(* IEC 61131-3 sources: sistemas-de-automacao/, 39 files *)

(* ---- E_PRODUCT_TYPE (DUT).st ---- *)
{attribute 'qualified_only'}
{attribute 'strict'}

// Enum para os tipos de itens que podem ser gerados e identificados no início da operação

TYPE E_PRODUCT_TYPE :
(
	e_productType_unknown := 0, // Caso o item ainda não tenha sido identificado ou tenha ocorrido algum erro
								// durante a identificação
	e_productType_plastic := 1, // Caso o item seja um bloco de plástico
	e_productType_metal := 2, // Caso o item seja um bloco de metal
	e_productType_box := 3 // Caso o item seja uma caixa
);
END_TYPE

(* ---- ST_PRODUCT (DUT).st ---- *)
TYPE ST_PRODUCT :

// Struct que guarda as informações sobre um produto, como o tipo dele, se ele já foi processado ou se ele é metálico
// Na prática só foi usada a informação de se o produto é metálico ou não, mas caso o projeto necessitasse de mais
// features ou fosse expandido de alguma forma, a struct permitiria essas expansão sem muito retrabalho

STRUCT
	productType : E_PRODUCT_TYPE;
	processed : BOOL;
	metal : BOOL;
END_STRUCT
END_TYPE

(* ---- ST_PRODUCT.DUT ---- *)
TYPE ST_PRODUCT :
STRUCT
	productType : E_PRODUCT_TYPE;
	metal       :           BOOL;
	processed   :           BOOL;

END_STRUCT
END_TYPE

(* ---- ST_PRODUCT.st ---- *)
TYPE ST_PRODUCT :
STRUCT
	productType : E_PRODUCT_TYPE;
	processed : BOOL;

END_STRUCT
END_TYPE

(* ---- ST_QUEUE.st ---- *)
TYPE ST_QUEUE :
STRUCT
 head : POINTER OF ST_QUEUE_ITEM;
 tail : POINTER OF ST_QUEUE_ITEM;
END_STRUCT
END_TYPE

(* ---- constante (GVL).st ---- *)
VAR_GLOBAL CONSTANT
    Xidle : INT := 500; // As coordenadas do Gantry CNC quando ele estiver ocioso
    Yidle : INT := 500;
    Zidle : INT := 200;

    XconveyorPlas : INT := 470; // As coordenadas do Gantry CNC para detectar uma caixa passando
    YconveyorPlas : INT := 600; // pela esteira de plástico usando o sensor SPP
    ZconveyorPlas : INT := 1000;

    XconveyorMetal : INT := 1000; // As coordenadas do Gantry CNC para detectar uma caixa passando
    YconveyorMetal : INT := 600;  // pela esteira de plástico usando o sensor SPP
    ZconveyorMetal : INT := 1000;

    Xpart : INT := 110; // As coordenadas do Gantry CNC para pegar uma peça na esteira da usinagem
    Ypart : INT := 500;
    Zpart : INT := 830;

    XboxMetal : INT := 850; // As coordenadas do Gantry CNC para pôr uma peça numa caixa da esteira
    YboxMetal : INT := 500; // de metal
    ZboxMetal : INT := 800;

    XboxPlas : INT := 330; // As coordenadas do Gantry CNC para pôr uma peça numa caixa da esteira
    YboxPlas : INT := 500; // de plástico
    ZboxPlas : INT := 800;

END_VAR

(* ---- constante.VAR ---- *)
{attribute 'qualified_only'}
VAR_GLOBAL CONSTANT
    Xidle : INT := 500;
    Yidle : INT := 500;
    Zidle : INT := 200;

    XconveyorPlas : INT := 470;
    YconveyorPlas : INT := 600;
    ZconveyorPlas : INT := 1000;

    XconveyorMetal : INT := 1000;
    YconveyorMetal : INT := 600;
    ZconveyorMetal : INT := 1000;

    Xpart : INT := 110;
    Ypart : INT := 500;
    Zpart : INT := 830;

    XboxMetal : INT := 850;
    YboxMetal : INT := 500;
    ZboxMetal : INT := 800;

    XboxPlas : INT := 330;
    YboxPlas : INT := 500;
    ZboxPlas : INT := 800;

END_VAR

(* ---- FIO (GVL).st ---- *)
{attribute 'qualified_only'}
VAR_GLOBAL
    i_DS2        			  		: BOOL; // Sensor óptico da balança
    i_Emergencia              		: BOOL; // Botão de emergência
	i_MachiningCenterOpened   		: BOOL; // Centro de usinagem livre
	i_MachiningCenterIsBusy   		: BOOL; // Centro de usinagem trabalhando
	i_MachiningCenterHasError 		: BOOL; // Erro no processo de usinagem
	i_RS1 					  		: BOOL; // Sensor óptico da usinagem
	i_RS2 					  		: BOOL; // Sensor óptico do empacotamento
	i_SC    				  		: BOOL; // Sensor capacitivo
	i_SC1Mais 				  		: BOOL; // Fim de curso do pistão - estendido
	i_SC1Menos 	 			  		: BOOL; // Fim de curso do pistão - retraido
    i_SI        			  		: BOOL; // Sensor indutivo
	i_SP 					  		:  INT; // Sensor da balança (4.0 plástico; 5.0 metal; 1.5 caixa)
	i_SPMais 				  		: BOOL; // Botão de aumentar quantidade de itens por caixa
	i_SPMenos 				  		: BOOL; // Botão de diminuir quantidade de itens por caixa
	i_SPP 					  		: BOOL; // Sensor de item pego pela ponte CNC
	i_Start 				  		: BOOL; // Botão START
	i_Stop 					  		: BOOL; // Botão STOP
    i_XPOS        			  		:  INT; // Dado da posição X atual da ponte CNC
    i_YPOS    				  		:  INT; // Dado da posição Y atual da ponte CNC
    i_ZPOS      			  		:  INT; // Dado da posição Z atual da ponte CNC
	i_DS3        			  		: BOOL; // Sensor óptico da esteira de plástico
	i_DS4        			  		: BOOL; // Sensor óptico da esteira de metal

	o_C1 					  		: BOOL; // Pistão
	o_Caixas_Emissor_1 		  		: BOOL; // Emissor de caixas (metal)
	o_E1 					  		: BOOL; // Primeira Esteira do classificador
	o_E2 					  		: BOOL; // Esteira final do classificador e inicial da usinagem
	o_E3 					  		: BOOL; // Esteira inicial do empacotamento
	o_EMETAL1 				  		: BOOL; // Primeira esteira de rolo do empacotamento de metal
	o_EMETAL2 				  		: BOOL; // Segunda esteira de rolo do empacotamento de metal
	o_EMETAL3 				  		: BOOL; // Terceira esteira de rolo do empacotamento de metal
	o_Emissor_Partes 		  		: BOOL; // Emissor dos itens (Deixar ligado)
	o_Emitter_4 			  		: BOOL; // Emissor de caixas (plástico)
	o_EPLASTIC1 			  		: BOOL; // Primeira esteira de rolo do empacotamento de plástico
	o_EPLASTIC2 			  		: BOOL; // Segunda esteira de rolo do empacotamento de plástico
	o_EPLASTIC3 			  	   	: BOOL; // Terceira esteira de rolo do empacotamento de plástico
	o_E_SP 					  	   	: BOOL; // Esteira da balança
	o_LedG 					  	   	: BOOL; // Led verde no canto da usinagem
	o_LedR 					  	   	: BOOL; // Led vermelho no canto da usinagem
	o_LedSPMais 			  	   	: BOOL; // Led do botão SP+
	o_LedSPMenos 			  	   	: BOOL; // Led do botão SP-
	o_LedStart 				  	   	: BOOL; // Led do botão START
	o_LedStop 				  	   	: BOOL; // Led do botão STOP
	o_LedY 					  	   	: BOOL; // Led amarelo no canto da usinagem
    o_RB1_Stop 				  	   	: BOOL; // Botão de interrupção do processo do braço robótico + usinagem
	o_RB1_Reset 			  	   	: BOOL; // Botão de reset do processo do braço robótico + usinagem
	o_RB1_Start 			  	  	: BOOL; // Botão de iniciar o processo do braço robótico + usinagem
	o_Succao 				  	  	: BOOL; // Acionamento da sucção da ponte CNC
    o_X           			  		:  INT; // Posição X da ponte CNC
    o_Y   					  		:  INT; // Posição Y da ponte CNC
    o_Z  					  		:  INT; // Posição Z da ponte CNC
	o_MachiningCenterProduceLids    : BOOL; // Modo de usinagem do plástico
	o_NumCaixas               		:  INT;  // Número de caixas
	o_NumMetal                		:  INT;  // Número de itens de metal
	o_NumPlastico             		:  INT;  // Número de itens de plástico
END_VAR

(* ---- FIO.VAR ---- *)
{attribute 'qualified_only'}
VAR_GLOBAL
    i_DS2        			  : BOOL; // Sensor óptico da balança
    i_Emergencia              : BOOL; // Botão de emergência
	i_MachiningCenterOpened   : BOOL; // Centro de usinagem livre
	i_MachiningCenterIsBusy   : BOOL; // Centro de usinagem trabalhando
	i_MachiningCenterHasError : BOOL; // Erro no processo de usinagem
	i_RS1 					  : BOOL; // Sensor óptico da usinagem
	i_RS2 					  : BOOL; // Sensor óptico do empacotamento
	i_SC    				  : BOOL; // Sensor capacitivo
	i_SC1Mais 				  : BOOL; // Fim de curso do pistão - estendido
	i_SC1Menos 	 			  : BOOL; // Fim de curso do pistão - retraido
    i_SI        			  : BOOL; // Sensor indutivo
	i_SP 					  : REAL; // Sensor da balança (4.0 plástico; 5.0 metal; 1.5 caixa)
	i_SPMais 				  : BOOL; // Botão de aumentar quantidade de itens por caixa
	i_SPMenos 				  : BOOL; // Botão de diminuir quantidade de itens por caixa
	i_SPP 					  : BOOL; // Sensor de item pego pela ponte CNC
	i_Start 				  : BOOL; // Botão START
	i_Stop 					  : BOOL; // Botão STOP
    i_XPOS        			  : REAL; // Dado da posição X atual da ponte CNC
    i_YPOS    				  : REAL; // Dado da posição Y atual da ponte CNC
    i_ZPOS      			  : REAL; // Dado da posição Z atual da ponte CNC

	o_C1 					  : BOOL; // Pistão
	o_Caixas_Emissor_1 		  : BOOL; // Emissor de caixas (metal)
	o_E1 					  : BOOL; // Primeira Esteira do classificador
	o_E2 					  : BOOL; // Esteira final do classificador e inicial da usinagem
	o_E3 					  : BOOL; // Esteira inicial do empacotamento
	o_EMETAL1 				  : BOOL; // Primeira esteira de rolo do empacotamento de metal
	o_EMETAL2 				  : BOOL; // Segunda esteira de rolo do empacotamento de metal
	o_EMETAL3 				  : BOOL; // Terceira esteira de rolo do empacotamento de metal
	o_Emissor_Partes 		  : BOOL; // Emissor dos itens (Deixar ligado)
	o_Emitter_4 			  : BOOL; // Emissor de caixas (plástico)
	o_EPLASTIC1 			  : BOOL; // Primeira esteira de rolo do empacotamento de plástico
	o_EPLASTIC2 			  : BOOL; // Segunda esteira de rolo do empacotamento de plástico
	o_EPLASTIC3 			  : BOOL; // Terceira esteira de rolo do empacotamento de plástico
	o_E_SP 					  : BOOL; // Esteira da balança
	o_LedG 					  : BOOL; // Led verde no canto da usinagem
	o_LedR 					  : BOOL; // Led vermelho no canto da usinagem
	o_LedSPMais 			  : BOOL; // Led do botão SP+
	o_LedSPMenos 			  : BOOL; // Led do botão SP-
	o_LedStart 				  : BOOL; // Led do botão START
	o_LedStop 				  : BOOL; // Led do botão STOP
	o_LedY 					  : BOOL; // Led amarelo no canto da usinagem
    o_RB1_Stop 				  : BOOL; // Botão de interrupção do processo do braço robótico + usinagem
	o_RB1_Reset 			  : BOOL; // Botão de reset do processo do braço robótico + usinagem
	o_RB1_Start 			  : BOOL; // Botão de iniciar o processo do braço robótico + usinagem
	o_Succao 				  : BOOL; // Acionamento da sucção da ponte CNC
    o_X           			  : REAL; // Posição X da ponte CNC
    o_Y   					  : REAL; // Posição Y da ponte CNC
    o_Z  					  : REAL; // Posição Z da ponte CNC
END_VAR

(* ---- global (GVL).st ---- *)
{attribute 'qualified_only'}
VAR_GLOBAL
	// Filas de itens
	Fila_cla : FB_PRODUCT_QUEUE; // Fila da máquina de estados da classificação
	Fila_usi : FB_PRODUCT_QUEUE; // Fila da máquina de estados da usinagem
	Fila_emp : FB_PRODUCT_QUEUE; // Fila da máquina de estados do empacotamento
END_VAR

(* ---- global.VAR ---- *)
{attribute 'qualified_only'}
VAR_GLOBAL
	// Filas de itens
	Fila_cla : FB_PRODUCT_QUEUE;
	Fila_usi : FB_PRODUCT_QUEUE;
	Fila_emp : FB_PRODUCT_QUEUE;
END_VAR

(* ---- GLOBAL_VAR.VAR ---- *)
{attribute 'qualified_only'}
VAR_GLOBAL
    i_DS2        : BOOL;
    i_Emergencia         : BOOL;
	i_MachiningCenterOpened : BOOL;
	i_MachiningCenterIsBusy : BOOL;
	i_MachiningCenterHasError : BOOL;
	i_RS1 : BOOL;
	i_RS2 : BOOL;
	i_SC    : BOOL;
	i_SC1Mais : BOOL;
	i_SC1Menos : BOOL;
    i_SI        : BOOL;
	i_SP : REAL;
	i_SPMais : BOOL;
	i_SPMenos : BOOL;
	i_SPP : BOOL;
	i_Start : BOOL;
	i_Stop : BOOL;
    i_XPOS        : REAL;
    i_YPOS    : REAL;
    i_ZPOS      : REAL;

    o_RB1 : BOOL;
    o_E1  : BOOL;
    o_E2           : BOOL;
    o_E3         : BOOL;
    o_X           : REAL;
    o_Y   : REAL;
    o_Z  : REAL;
END_VAR

(* ---- pushFilaEmp (FUN).st ---- *)
FUNCTION pushFilaEmp : BOOL
VAR_INPUT
END_VAR
VAR
END_VAR

global.Fila_emp.itemIn.metal := global.Fila_usi.itemOut.metal; // Seta o item que está entrando na fila de
                                                               // empacotamento igual ao item que está saindo
                                                               // da fila de usinagem
global.Fila_emp(push := TRUE);  // Dá push na fila de empacotamento
global.Fila_emp(push := FALSE);
global.Fila_usi(pop := TRUE);  // Dá pop na fila de usinagem
global.Fila_usi(pop := FALSE);

(* ---- pushFilaEmp.FUN ---- *)
FUNCTION pushFilaEmp : BOOL
VAR_INPUT
END_VAR
VAR
END_VAR

global.Fila_emp.itemIn := global.Fila_usi.itemOut;
global.Fila_emp(push := TRUE);
global.Fila_emp.push := FALSE;
global.Fila_usi(pop := TRUE);
global.Fila_usi.pop := FALSE;

(* ---- pushFilaUsi (FUN).st ---- *)
FUNCTION pushFilaUsi : BOOL
VAR_INPUT
END_VAR
VAR
END_VAR

global.Fila_usi.itemIn.metal := global.Fila_cla.itemOut.metal; // Seta o item que está entrando na fila de
                                                               // usinagem igual ao item que está saindo
                                                               // da fila de classificação
global.Fila_usi(push := TRUE);  // Dá push na fila de usinagem
global.Fila_usi(push := FALSE);
global.Fila_cla(pop := TRUE);   // Dá pop na fila de classificação
global.Fila_cla(pop := FALSE);

(* ---- pushFilaUsi.FUN ---- *)
FUNCTION pushFilaUsi : BOOL
VAR_INPUT
END_VAR
VAR
END_VAR

global.Fila_usi.itemIn.metal := global.Fila_cla.itemOut.metal;
global.Fila_usi(push := TRUE);
global.Fila_usi(push := FALSE);
global.Fila_cla(pop := TRUE);
global.Fila_cla(pop := FALSE);

(* ---- registrarItem (FUN).st ---- *)
FUNCTION registrarItem : BOOL
VAR_INPUT
END_VAR
VAR
END_VAR

global.Fila_cla.itemIn.metal := FIO.i_SI; // Seta a variável metal do item de entrada da fila de classificação
                                          // como a informação indicada pelo sensor indutivo
global.Fila_cla(push := TRUE);  // Dá push na fila de classificação
global.Fila_cla(push := FALSE);

(* ---- registrarItem.FUN ---- *)
FUNCTION registrarItem : BOOL
VAR_INPUT
END_VAR
VAR
END_VAR

global.Fila_cla.itemIn.metal := FIO.i_SI;
global.Fila_cla(push := TRUE);
global.Fila_cla(push := FALSE);

(* ---- empurrarCaixa (FB).st ---- *)
FUNCTION_BLOCK empurrarCaixa
VAR_INPUT
    start   : BOOL; // Variável de entrada que em rising inicia o movimento
END_VAR

VAR_OUTPUT
    done  : BOOL; // Variável de saída que indica que o movimento foi concluído
END_VAR

VAR
	trigStart : R_TRIG;
    state : INT := 0;
END_VAR

trigStart(CLK:=start);

CASE state OF

    0: // Estado Ocioso
        IF trigStart.Q THEN
            state := 10;
			done := FALSE;
        END_IF

    10: // Move pistão para frente
        IF NOT FIO.i_SC1Mais THEN
            FIO.o_C1 := TRUE;
        ELSE
            state := 20;
        END_IF

    20: // Move pistão para trás
        IF NOT FIO.i_SC1Menos THEN
            FIO.o_C1 := FALSE;
        ELSE
            state := 30;
        END_IF

    30: // Finalizado
        done := TRUE;
		state := 0;

END_CASE

(* ---- empurrarCaixa.FB ---- *)
FUNCTION_BLOCK FB_PRODUCT_QUEUE
VAR_INPUT
    start   : BOOL;
END_VAR

VAR_OUTPUT
    done  : BOOL;
END_VAR

VAR
	trigStart : R_TRIG;
    state : INT := 0;
END_VAR

trigStart(CLK:=start);

CASE state OF

    0: // Idle
        IF trigStart.Q THEN
            state := 10;
			done := FALSE;
        END_IF

    10: // Move Forward
        IF NOT FIO.i_SC1Mais THEN
            FIO.o_C1 := TRUE;
        ELSE
            state := 20;
        END_IF

    20: // Move Back
        IF NOT FIO.i_SC1Menos THEN
            FIO.o_C1 := FALSE;
        ELSE
            state := 30;
        END_IF

    30: // Finalizado
        done := TRUE;
		state := 0;

END_CASE

(* ---- FB_MoveTo (FB).st ---- *)
FUNCTION_BLOCK FB_MoveTo
VAR_INPUT
    targetX : INT;    // Coordenadas da posição desejada
    targetY : INT;
    targetZ : INT;
    start   : BOOL;   // pulso de start
END_VAR

VAR_OUTPUT
    done : BOOL;      // TRUE quando chegou
END_VAR

VAR
	trigStart : R_TRIG;
    state : INT := 0;
	timer : TON;
END_VAR

trigStart(CLK:=start);

CASE state OF

    0: // Estado ocioso
        IF trigStart.Q THEN
            state := 10;
			done := FALSE;
        END_IF

    10: // Move no eixo X
		FIO.o_X := targetX;
        IF (FIO.i_XPOS < targetX - 5) OR (FIO.i_XPOS > targetX + 5) THEN // Deixa um intervalo de +/- 5 para o sensor de posição
            FIO.o_X := targetX;
        ELSE
            state := 20;
        END_IF

    20: // Move no eixo Y
	FIO.o_Y := targetY;
        IF (FIO.i_YPOS < targetY - 5) OR (FIO.i_YPOS > targetY + 5) THEN
            FIO.o_Y := targetY;
        ELSE
            state := 30;
        END_IF

    30: // Move no eixo Z
	FIO.o_Z := targetZ;
        IF (FIO.i_ZPOS < targetZ - 5) OR (FIO.i_ZPOS > targetZ + 5) THEN
            FIO.o_Z := targetZ;
        ELSE
            state := 40;
        END_IF

    40: // Finalizado
	Timer(IN:=TRUE, PT:=T#0.5S);
	IF Timer.Q THEN
		Timer.IN := FALSE;
        done := TRUE;
		state := 0;
	END_IF;

END_CASE

(* ---- FB_MoveTo.FB ---- *)
FUNCTION_BLOCK FB_MoveTo
VAR_INPUT
    targetX : INT;
    targetY : INT;
    targetZ : INT;
    start   : BOOL;   // pulso de start
END_VAR

VAR_OUTPUT
    done : BOOL;      // TRUE quando chegou
END_VAR

VAR
	trigStart : R_TRIG;
    state : INT := 0;
END_VAR

trigStart(CLK:=start);

CASE state OF

    0: // Idle
        IF trigStart.Q THEN
            state := 10;
			done := FALSE;
        END_IF

    10: // Move X
        IF (FIO.i_XPOS < targetX - 10) OR (FIO.i_XPOS > targetX + 10) THEN
            FIO.o_X := targetX;
        ELSE
            state := 20;
        END_IF

    20: // Move Y
        IF (FIO.i_YPOS < targetY - 10) OR (FIO.i_YPOS > targetY + 10) THEN
            FIO.o_Y := targetY;
        ELSE
            state := 30;
        END_IF

    30: // Move Z
        IF (FIO.i_ZPOS < targetZ - 10) OR (FIO.i_ZPOS > targetZ + 10) THEN
            FIO.o_Z := targetZ;
        ELSE
            state := 40;
        END_IF

    40: // Finalizado
        done := TRUE;
		state := 0;

END_CASE

(* ---- FB_PRODUCT_QUEUE (FB).st ---- *)
FUNCTION_BLOCK FB_PRODUCT_QUEUE
VAR_INPUT
<<<<<<< HEAD:FB_PRODUCT_QUEUE (FB).st
    push : BOOL; // Sinais de entrada que determinam o método chamado do objeto
    pop  : BOOL;
    clear  : BOOL;
    itemIn : ST_PRODUCT; // Buffer do produto que vai entrar na fila
=======
    push : BOOL := FALSE;
    pop  : BOOL := FALSE;
    clear  : BOOL := FALSE;
    itemIn : ST_PRODUCT;
>>>>>>> origin/main:FB_PRODUCT_QUEUE.FB
END_VAR

VAR_OUTPUT
    itemOut : ST_PRODUCT; // Buffer do produto que vai sair da fila
    isEmpty : BOOL; // Informação se a fila está vazia
    isFull  : BOOL; // Informação se a fila está cheia
END_VAR

VAR
    // Triggers dos métodos
	trigPush : R_TRIG;
    trigPop  : R_TRIG;
    trigClear : R_TRIG;

    // Array que guarda de fato a informação dos produtos na fila
    buffer : ARRAY[1..100] OF ST_PRODUCT;
    head   : INT := 1; // Índice que indica o produto que está saindo da fila
    tail   : INT := 1; // Índice que indica o produto que está entrando na fila
    count  : INT := 0; // Quantidade de itens atualmente na fila
END_VAR

// Atualiza os detectores de flanco
trigPush(CLK := push);
trigPop(CLK := pop);
trigClear(CLK := clear);

// Peek
itemOut := buffer[head];

// Clear
IF trigClear.Q THEN
    head := 1;
    tail := head;
    count := 0;

// Dequeue
ELSIF trigPop.Q AND (count > 0) THEN
    head := (head MOD 100) + 1;
    count := count - 1;

// Enqueue
ELSIF trigPush.Q AND (count < 100) THEN
    buffer[tail] := itemIn;
    tail := (tail MOD 100) + 1;
    count := count + 1;
END_IF;

isEmpty := (count = 0);
isFull  := (count = 100);

(* ---- FB_PRODUCT_QUEUE.FB ---- *)
FUNCTION_BLOCK FB_PRODUCT_QUEUE
VAR_INPUT
    push : BOOL;
    pop  : BOOL;
    clear  : BOOL;
    itemIn : ST_PRODUCT;
END_VAR

VAR_OUTPUT
    itemOut : ST_PRODUCT;
    isEmpty : BOOL;
    isFull  : BOOL;
END_VAR

VAR
	trigPush : R_TRIG;
    trigPop  : R_TRIG;
    trigClear : R_TRIG;

    buffer : ARRAY[1..100] OF ST_PRODUCT;
    head   : INT := 1;
    tail   : INT := 1;
    count  : INT := 0;
END_VAR

// Atualiza os detectores de flanco
trigPush(CLK := push);
trigPop(CLK := pop);
trigClear(CLK := clear);

// Peek
itemOut := buffer[head];

// Clear
IF trigClear.Q THEN
    head := 1;
    tail := head;
    count := 0;

// Dequeue
ELSIF trigPop THEN
    head := (head MOD 100) + 1;
    count := count - 1;

// Enqueue
ELSIF trigPush AND (count < 100) THEN
    buffer[tail] := itemIn;
    tail := (tail MOD 100) + 1;
    count := count + 1;
END_IF;

isEmpty := (count = 0);
isFull  := (count = 100);

(* ---- moverMetal (FB).st ---- *)
FUNCTION_BLOCK moverMetal
VAR_INPUT
    start   : BOOL;   // pulso de start
END_VAR

VAR_OUTPUT
    done : BOOL;      // TRUE quando chegou
END_VAR

VAR
    empCNC : FB_MoveTo;
	trigStart : R_TRIG;
    state : INT := 0;

END_VAR

trigStart(CLK:=start);

CASE state OF

    0: // Estado ocioso
        IF trigStart.Q THEN
            state := 10;
			done := FALSE;
        END_IF

    10: // Move até o item
        empCNC(targetX := constante.Xpart, targetY := constante.Ypart, targetZ := constante.Zpart, start := TRUE);
        IF empCNC.done THEN
            empCNC(start := FALSE);
            state := 20;
        END_IF

    20: // Pega o item
        FIO.o_Succao := TRUE;
        IF FIO.i_SPP THEN
            state := 30;
        END_IF

    30: // Move para cima
        empCNC(targetX := constante.Xpart, targetY := constante.Ypart, targetZ := constante.Zpart - 50, start := TRUE);
        IF empCNC.done THEN
            empCNC(start := FALSE);
            state := 40;
        END_IF

    40: // Move até a caixa
        empCNC(targetX := constante.XboxMetal, targetY := constante.YboxMetal, targetZ := constante.ZboxMetal, start := TRUE);
        IF empCNC.done THEN
            empCNC(start := FALSE);
            state := 50;
        END_IF

    50: // Solta a peça
        FIO.o_Succao := FALSE;
        IF NOT FIO.i_SPP THEN
            state := 60;
        END_IF

    60: // Retorna a posição de descanso
        empCNC(targetX := constante.Xidle, targetY := constante.Yidle, targetZ := constante.Zidle, start := TRUE);
        IF empCNC.done THEN
            empCNC(start := FALSE);
            state := 70;
        END_IF

    70: // Finalizado
        done := TRUE;
		state := 0;

END_CASE

(* ---- moverMetal.FB ---- *)
FUNCTION_BLOCK moverMetal
VAR_INPUT
    start   : BOOL;   // pulso de start
END_VAR

VAR_OUTPUT
    done : BOOL;      // TRUE quando chegou
END_VAR

VAR
    empCNC : FB_MoveTo;
	trigStart : R_TRIG;
    state : INT := 0;

END_VAR

trigStart(CLK:=start);

CASE state OF

    0: // Idle
        IF trigStart.Q THEN
            state := 10;
			done := FALSE;
        END_IF

    10: // Move to part
        empCNC(targetX := constante.Xpart, targetY := constante.Ypart, targetZ := constante.Zpart, start := TRUE);
        IF empCNC.done THEN
            empCNC(start := FALSE);
            state := 20;
        END_IF

    20: // Catch part
        FIO.o_Succao := TRUE;
        IF FIO.i_SPP THEN
            state := 30;
        END_IF

    30: // Move Vertically
        empCNC(targetX := constante.Xpart, targetY := constante.Ypart, targetZ := constante.Zpart - 50, start := TRUE);
        IF empCNC.done THEN
            empCNC(start := FALSE);
            state := 40;
        END_IF

    40: // Move to box
        empCNC(targetX := constante.XboxMetal, targetY := constante.YboxMetal, targetZ := constante.ZboxMetal, start := TRUE);
        IF empCNC.done THEN
            empCNC(start := FALSE);
            state := 50;
        END_IF

    50: // Drop part off
        FIO.o_Succao := FALSE;
        IF NOT FIO.i_SPP THEN
            state := 60;
        END_IF

    60: // Return to idle position
        empCNC(targetX := constante.Xidle, targetY := constante.Yidle, targetZ := constante.Zidle, start := TRUE);
        IF empCNC.done THEN
            empCNC(start := FALSE);
            state := 70;
        END_IF

    70: // Finalizado
        done := TRUE;
		state := 0;

END_CASE

(* ---- moverPlastico (FB).st ---- *)
FUNCTION_BLOCK moverPlastico
VAR_INPUT
    start   : BOOL;  // pulso de start
END_VAR

VAR_OUTPUT
    done : BOOL;      // TRUE quando chegou
END_VAR

VAR
    empCNC : FB_MoveTo;
	trigStart : R_TRIG;
    state : INT := 0;

END_VAR

trigStart(CLK:=start);

CASE state OF

    0: // Estado ocioso
        IF trigStart.Q THEN
            state := 10;
			done := FALSE;
        END_IF

    10: // Move até o item
        empCNC(targetX := constante.Xpart, targetY := constante.Ypart, targetZ := constante.Zpart, start := TRUE);
        IF empCNC.done THEN
            empCNC(start := FALSE);
            state := 20;
        END_IF

    20: // Pega o item
        FIO.o_Succao := TRUE;
        IF FIO.i_SPP THEN
            state := 30;
        END_IF

    30: // Move para cima
        empCNC(targetX := constante.Xpart, targetY := constante.Ypart, targetZ := constante.Zpart - 50, start := TRUE);
        IF empCNC.done THEN
            empCNC(start := FALSE);
            state := 40;
        END_IF

    40: // Move até a caixa
        empCNC(targetX := constante.XboxPlas, targetY := constante.YboxPlas, targetZ := constante.ZboxPlas, start := TRUE);
        IF empCNC.done THEN
            empCNC(start := FALSE);
            state := 50;
        END_IF

    50: // Solta a peça
        FIO.o_Succao := FALSE;
        IF NOT FIO.i_SPP THEN
            state := 60;
        END_IF

    60: // Retorna a posição de descanso
        empCNC(targetX := constante.Xidle, targetY := constante.Yidle, targetZ := constante.Zidle, start := TRUE);
        IF empCNC.done THEN
            empCNC(start := FALSE);
            state := 70;
        END_IF

    70: // Finalizado
        done := TRUE;
		state := 0;

END_CASE

(* ---- moverPlastico.FB ---- *)
FUNCTION_BLOCK moverPlastico
VAR_INPUT
    start   : BOOL;  // pulso de start
END_VAR

VAR_OUTPUT
    done : BOOL;      // TRUE quando chegou
END_VAR

VAR
    empCNC : FB_MoveTo;
	trigStart : R_TRIG;
    state : INT := 0;

    // Coordenadas
    Xpart : INT := 0;
    Ypart : INT := 500;
    Zpart : INT := 850;
    Xbox : INT := 330;
    Ybox : INT := 500;
    Zbox : INT := 800;
    Xidle : INT := 500;
    Yidle : INT := 500;
    Zidle : INT := 50;

END_VAR

trigStart(CLK:=start);

CASE state OF

    0: // Idle
        IF trigStart.Q THEN
            state := 10;
			done := FALSE;
        END_IF

    10: // Move to part
        empCNC(targetX := Xpart, targetY := Ypart, targetZ := Zpart, start := TRUE);
        IF empCNC.done THEN
            empCNC(start := FALSE);
            state := 20;
        END_IF

    20: // Catch part
        FIO.o_Succao := TRUE;
        IF FIO.i_SPP THEN
            state := 30;
        END_IF

    30: // Move Vertically
        empCNC(targetX := Xpart, targetY := Ypart, targetZ := Zpart - 50, start := TRUE);
        IF empCNC.done THEN
            empCNC(start := FALSE);
            state := 40;
        END_IF

    40: // Move to box
        empCNC(targetX := Xbox, targetY := Ybox, targetZ := Zbox, start := TRUE);
        IF empCNC.done THEN
            empCNC(start := FALSE);
            state := 50;
        END_IF

    50: // Drop part off
        FIO.o_Succao := FALSE;
        IF NOT FIO.i_SPP THEN
            state := 60;
        END_IF

    60: // Return to idle position
        empCNC(targetX := Xidle, targetY := Yidle, targetZ := Zidle, start := TRUE);
        IF empCNC.done THEN
            empCNC(start := FALSE);
            state := 70;
        END_IF

    70: // Finalizado
        done := TRUE;
		state := 0;

END_CASE

(* ---- posicionarEsteiraMetal (FB).st ---- *)
FUNCTION_BLOCK posicionarEsteiraMetal
VAR_INPUT
    start   : BOOL;  // pulso de start
END_VAR

VAR_OUTPUT
    done : BOOL;      // TRUE quando chegou
END_VAR

VAR
	trigStart : R_TRIG;
	trigSensor : R_TRIG;
    state : INT := 0;

END_VAR

trigStart(CLK:=start);

CASE state OF

    0: // Estado ocioso
        IF trigStart.Q THEN
            state := 10;
			done := FALSE;
        END_IF

    10: // Liga as esteiras
        FIO.o_EMETAL1 := TRUE;
        FIO.o_EMETAL2 := TRUE;
        FIO.o_EMETAL3 := TRUE;
        state := 20;

    20: // Aguarda pelo trigger do sensor
        trigSensor(CLK:=FIO.i_DS4);
        IF trigSensor.Q THEN
            state := 30;
        END_IF

    30: // Desliga as esteiras
        FIO.o_EMETAL1 := FALSE;
        FIO.o_EMETAL2 := FALSE;
        FIO.o_EMETAL3 := FALSE;
        state := 40;

    40: // Finalizado
        done := TRUE;
		state := 0;

END_CASE

(* ---- posicionarEsteiraMetal.FB ---- *)
FUNCTION_BLOCK posicionarEsteiraMetal
VAR_INPUT
    start   : BOOL;  // pulso de start
END_VAR

VAR_OUTPUT
    done : BOOL;      // TRUE quando chegou
END_VAR

VAR
    empCNC : FB_MoveTo;
	trigStart : R_TRIG;
	trigSensor : R_TRIG;
    state : INT := 0;

    // Coordenadas
    Xconveyor : INT := 1000;
    Yconveyor : INT := 600;
    Zconveyor : INT := 990;
    Xidle : INT := 500;
    Yidle : INT := 500;
    Zidle : INT := 200;

END_VAR

trigStart(CLK:=start);

CASE state OF

    0: // Idle
        IF trigStart.Q THEN
            state := 10;
			done := FALSE;
        END_IF

    10: // Move to conveyor position
        empCNC(targetX := Xconveyor, targetY := Yconveyor, targetZ := Zconveyor, start := TRUE);
        IF empCNC.done THEN
            empCNC(start := FALSE);
            state := 20;
        END_IF

    20: // Turn on conveyor
        FIO.o_EMETAL1 := TRUE;
        FIO.o_EMETAL2 := TRUE;
        FIO.o_EMETAL3 := TRUE;
        state := 30;

    30: // Wait for trigger
        trigSensor(CLK:=FIO.i_SPP);
        IF trigSensor.Q THEN
            state := 40;
        END_IF

    40: // Turn off conveyor
        FIO.o_EMETAL1 := FALSE;
        FIO.o_EMETAL2 := FALSE;
        FIO.o_EMETAL3 := FALSE;
        state := 50;

    50: // Return to idle position
        empCNC(targetX := Xidle, targetY := Yidle, targetZ := Zidle, start := TRUE);
        IF empCNC.done THEN
            empCNC(start := FALSE);
            state := 60;
        END_IF

    60: // Finalizado
        done := TRUE;
		state := 0;

END_CASE

(* ---- posicionarEsteiraPlastico (FB).st ---- *)
FUNCTION_BLOCK posicionarEsteiraPlastico
VAR_INPUT
    start   : BOOL;  // pulso de start
END_VAR

VAR_OUTPUT
    done : BOOL;      // TRUE quando chegou
END_VAR

VAR
	trigStart : R_TRIG;
	trigSensor : R_TRIG;
    state : INT := 0;

END_VAR

trigStart(CLK:=start);

CASE state OF

    0: // Estado ocioso
        IF trigStart.Q THEN
            state := 10;
			done := FALSE;
        END_IF

    10: // Liga as esteiras
        FIO.o_EPLASTIC1 := TRUE;
        FIO.o_EPLASTIC2 := TRUE;
        FIO.o_EPLASTIC3 := TRUE;
        state := 20;

    20: // Aguarda pelo trigger do sensor
        trigSensor(CLK:=FIO.i_DS3);
        IF trigSensor.Q THEN
            state := 30;
        END_IF

    30: // Desliga as esteiras
        FIO.o_EPLASTIC1 := FALSE;
        FIO.o_EPLASTIC2 := FALSE;
        FIO.o_EPLASTIC3 := FALSE;
        state := 40;

    40: // Finalizado
        done := TRUE;
		state := 0;

END_CASE

(* ---- posicionarEsteiraPlastico.FB ---- *)
FUNCTION_BLOCK posicionarEsteiraPlastico
VAR_INPUT
    start   : BOOL;  // pulso de start
END_VAR

VAR_OUTPUT
    done : BOOL;      // TRUE quando chegou
END_VAR

VAR
    empCNC : FB_MoveTo;
	trigStart : R_TRIG;
	trigSensor : R_TRIG;
    state : INT := 0;

    // Coordenadas
    Xconveyor : INT := 470;
    Yconveyor : INT := 600;
    Zconveyor : INT := 1000;

    Xidle : INT := 500;
    Yidle : INT := 500;
    Zidle : INT := 200;

END_VAR

trigStart(CLK:=start);

CASE state OF

    0: // Idle
        IF trigStart.Q THEN
            state := 10;
			done := FALSE;
        END_IF

    10: // Move to conveyor position
        empCNC(targetX := constante.XconveyorPlas, targetY := constante.YconveyorPlas, targetZ := constante.ZconveyorPlas, start := TRUE);
        IF empCNC.done THEN
            empCNC(start := FALSE);
            state := 20;
        END_IF

    20: // Turn on conveyor
        FIO.o_EPLASTIC1 := TRUE;
        FIO.o_EPLASTIC2 := TRUE;
        FIO.o_EPLASTIC3 := TRUE;
        state := 30;

    30: // Wait for trigger
        trigSensor(CLK:=FIO.i_SPP);
        IF trigSensor.Q THEN
            state := 40;
        END_IF

    40: // Turn off conveyor
        FIO.o_EPLASTIC1 := FALSE;
        FIO.o_EPLASTIC2 := FALSE;
        FIO.o_EPLASTIC3 := FALSE;
        state := 50;

    50: // Return to idle position
        empCNC(targetX := constante.Xidle, targetY := constante.Yidle, targetZ := constante.Zidle, start := TRUE);
        IF empCNC.done THEN
            empCNC(start := FALSE);
            state := 60;
        END_IF

    60: // Finalizado
        done := TRUE;
		state := 0;

END_CASE

(* ---- pushFilaEmp.FB ---- *)
FUNCTION_BLOCK pushFilaEmp // TODO - Substitua esse Function Block por uma função, se baseie na função registrarItem, essa função está funcionando bem

VAR_INPUT
    start   : BOOL;   // pulso de start
END_VAR

VAR_OUTPUT
    done : BOOL;      // TRUE quando chegou
END_VAR

VAR
	trigStart : R_TRIG;
    state : INT := 0;
    popTimer : TON := (PT := T#0.1S);

END_VAR

trigStart(CLK:=start);

CASE state OF

    0: // Idle
        IF trigStart.Q THEN
            state := 10;
			done := FALSE;
        END_IF

    10: // Push item into emp queue
		global.Fila_emp(push := FALSE);
        global.Fila_emp(push := TRUE, itemIn := global.Fila_usi.itemOut);
        IF (global.Fila_emp.itemOut.metal = global.Fila_usi.itemOut.metal) THEN
            state := 20;
        END_IF

    20: // Push item from usi queue
		global.Fila_usi(pop := FALSE);
        global.Fila_usi(pop := TRUE);
        popTimer(IN := TRUE);
        IF popTimer.Q THEN
			global.Fila_usi(pop := FALSE);
            popTimer(IN := FALSE);
            state := 30;
        END_IF

    30: // Finalizado
        done := TRUE;
		state := 0;

END_CASE

(* ---- pushFilaUsi.FB ---- *)
FUNCTION_BLOCK pushFilaUsi

VAR_INPUT
    start   : BOOL;   // pulso de start
END_VAR

VAR_OUTPUT
    done : BOOL;      // TRUE quando chegou
END_VAR

VAR
	trigStart : R_TRIG;
    state : INT := 0;
    popTimer : TON := (PT := T#0.1S);

END_VAR

trigStart(CLK:=start);

CASE state OF

    0: // Idle
        IF trigStart.Q THEN
            state := 10;
			done := FALSE;
        END_IF

    10: // Push item into usi queue
		global.Fila_usi(push := FALSE);
        global.Fila_usi(push := TRUE, itemIn := global.Fila_cla.itemOut);
        IF (global.Fila_usi.itemOut.metal = global.Fila_cla.itemOut.metal) THEN
            state := 20;
        END_IF

    20: // Push item from cla queue
		global.Fila_cla(pop := FALSE);
        global.Fila_cla(pop := TRUE);
        popTimer(IN := TRUE);
        IF popTimer.Q THEN
			global.Fila_cla(pop := FALSE);
            popTimer(IN := FALSE);
            state := 30;
        END_IF

    30: // Finalizado
        done := TRUE;
		state := 0;

END_CASE

(* ---- reposicionarEsteiraMetal.FB ---- *)
FUNCTION_BLOCK reposicionarEsteiraMetal
VAR_INPUT
    start   : BOOL;  // pulso de start
END_VAR

VAR_OUTPUT
    done : BOOL;      // TRUE quando chegou
END_VAR

VAR
    empCNC : FB_MoveTo;
    posicionarEstMetal : posicionarEsteiraMetal;
	trigStart : R_TRIG;
	trigSensor : R_TRIG;
    state : INT := 0;

END_VAR

trigStart(CLK:=start);

CASE state OF

    0: // Idle
        IF trigStart.Q THEN
            state := 10;
			done := FALSE;
        END_IF

    10: // Move to conveyor position
        empCNC(targetX := constante.XconveyorMetal, targetY := constante.YconveyorMetal, targetZ := constante.ZconveyorMetal, start := TRUE);
        IF empCNC.done THEN
            empCNC(start := FALSE);
            state := 20;
        END_IF

    20: // Turn on conveyor
        FIO.o_EMETAL1 := TRUE;
        FIO.o_EMETAL2 := TRUE;
        FIO.o_EMETAL3 := TRUE;
        state := 30;

    30: // Wait for trigger
        trigSensor(CLK:=FIO.i_SPP);
        IF trigSensor.Q THEN
            FIO.o_EMETAL1 := FALSE;
            FIO.o_EMETAL2 := FALSE;
            FIO.o_EMETAL3 := FALSE;
            state := 40;
        END_IF

    40: // call reposicionar FB
      	posicionarEstMetal(start:=TRUE);

      	// Transições de estado
      	IF posicionarEstMetal.done THEN
          posicionarEstMetal(start := FALSE);
      		state := 50;
      	END_IF;

    50: // Return to idle position
        empCNC(targetX := constante.Xidle, targetY := constante.Yidle, targetZ := constante.Zidle, start := TRUE);
        IF empCNC.done THEN
            empCNC(start := FALSE);
            state := 60;
        END_IF

    60: // Finalizado
        done := TRUE;
		state := 0;

END_CASE

(* ---- reposicionarEsteiraPlastico.FB ---- *)
FUNCTION_BLOCK reposicionarEsteiraPlastico
VAR_INPUT
    start   : BOOL;  // pulso de start
END_VAR

VAR_OUTPUT
    done : BOOL;      // TRUE quando chegou
END_VAR

VAR
    empCNC : FB_MoveTo;
    posicionarEstPlas : posicionarEsteiraPlastico;
	trigStart : R_TRIG;
	trigSensor : R_TRIG;
    state : INT := 0;

END_VAR

trigStart(CLK:=start);

CASE state OF

    0: // Idle
        IF trigStart.Q THEN
            state := 10;
			done := FALSE;
        END_IF

    10: // Move to conveyor position
        empCNC(targetX := constante.Xconveyor, targetY := constante.Yconveyor, targetZ := constante.Zconveyor, start := TRUE);
        IF empCNC1.done THEN
            empCNC(start := FALSE);
            state := 20;
        END_IF

    20: // Turn on conveyor
        FIO.o_EPLASTIC1 := TRUE;
        FIO.o_EPLASTIC2 := TRUE;
        FIO.o_EPLASTIC3 := TRUE;
        state := 30;

    30: // Wait for trigger
        trigSensor(CLK:=FIO.i_SPP);
        IF trigSensor.Q THEN
            FIO.o_EPLASTIC1 := FALSE;
            FIO.o_EPLASTIC2 := FALSE;
            FIO.o_EPLASTIC3 := FALSE;
            state := 40;
        END_IF

    40: // call reposicionar FB
      	posicionarEstPlas(start:=TRUE);

      	// Transições de estado
      	IF posicionarEstPlas.done THEN
          posicionarEstPlas(start := FALSE);
      		state := 50;
      	END_IF;

    50: // Return to idle position
        empCNC(targetX := constante.Xidle, targetY := constante.Yidle, targetZ := constante.Zidle, start := TRUE);
        IF empCNC.done THEN
            empCNC(start := FALSE);
            state := 60;
        END_IF

    60: // Finalizado
        done := TRUE;
		state := 0;

END_CASE

(* ---- PLC_PRG (PRG).st ---- *)
PROGRAM PLC_PRG
VAR
    // Estados das máquinas
    E_Cla : INT := 0;      		// Classificadora
	E_Cla_anterior : INT := 0; 	// Guarda o estado da máquina classificadora antes da espera
    E_Usi : INT := 0;      		// Usinagem
    E_Emp : INT := 0;      		// Empacotamento
    E_Sup : INT := 0;      		// Supervisora

	// Oneshot das máquinas
	os_cla : ARRAY[0..10] OF BOOL; // Classificação
	os_usi : ARRAY[0..10] OF BOOL; // Usinagem
	os_emp : ARRAY[0..10] OF BOOL; // Empacotamento
	os_sup : ARRAY[0..10] OF BOOL; // Supervisora

	os_reset : ARRAY[0..10] OF BOOL; // Array de reset dos oneshot

    // Entradas gerais
    START : BOOL;
    STOP  : BOOL;
	EMER  : BOOL;

    // Sinais de emergência
    Emergencia1 : BOOL := FALSE;
    Emergencia2 : BOOL := FALSE;
    Emergencia3 : BOOL := FALSE;

    // Comandos da máquina supervisora
    Maquina1 : BOOL := FALSE;   // Liga classificadora
    Maquina2 : BOOL := FALSE;   // Liga usinagem
    Maquina3 : BOOL := FALSE;   // Liga empacotamento

	// Comunicação entre máquinas
	esperaCla : BOOL := FALSE;  // Sinal que faz a máquina classificadora entrar em espera

    // Sensores
    SC  : BOOL := FALSE;    // Sensor capacitivo
	SI  : BOOL := FALSE;    // Sensor indutivo
    OP1 : BOOL := FALSE;    // Sensor óptico 1
    OP2 : BOOL := FALSE;    // Sensor óptico 2
    OP3 : BOOL := FALSE;    // Sensor óptico 3

    // Contadores
    contador_classificacao : INT := 0; // Itens que passaram pela classificação
    contador_usinagem      : INT := 0; // Itens que passaram pela usinagem
    contador_empacotamento : INT := 0; // Itens que passaram pelo empacotamento

    // Contadores da empacotadora
    plastico_counter : INT := 0; // Quantidade de itens de plástico na caixa de plástico atual
    metal_counter    : INT := 0; // Quantidade de itens de metal na caixa de metal atual
    itemPorCaixa     : INT := 3; // Quantidade de itens que devem ser colocados em uma caixa no empacotamento

    // Buffers de variáveis lógicas
	caixa    : BOOL; // Guarda a informação se o item em cima da balança é uma caixa ou não

	// Timers de emergência
	Timer_sc  	  : TON := (PT := T#30S);
	Timer_op1 	  : TON := (PT := T#30S);
	Timer_op2     : TON := (PT := T#30S);
<<<<<<< HEAD:PLC_PRG (PRG).st
<<<<<<< HEAD:PLC_PRG (PRG).st
=======
>>>>>>> 670f2d2 (Código funcionando 100% e com 100% de eficiência):PLC_PRG.st
	Timer_usi     : TON := (PT := T#15S);
	Timer_op3     : TON := (PT := T#40S);
=======
	Timer_op3     : TON := (PT := T#30S);
>>>>>>> 3a60cd6 (Update PLC_PRG.st):PLC_PRG.st

	// Delays
	delayEstabilizarBalanca : TON := (PT := T#1.5S); // Delay da balança

	// Triggers
	trigSC : R_TRIG; // Trigger ativo na subida do sensor SC,
					 // usado para identificar um item passando na classificação
	trigUsiConcluida : F_TRIG; // Trigger ativo na descida da variável MachiningCenterIsBusy,
							   // Usado para identificar quando a usinagem é concluída
	trigUsiOcupada : R_TRIG; // Trigger ativo na subida da variável MachiningCenterIsBusy,
							 // Usado para identificar quando a usinagem é iniciada
	trigSPMais : R_TRIG; // Triggers de subida dos botões SP+ e SP-, usado para identificar
	trigSPMenos : R_TRIG; // quando esse botões são pressionados

	// Blocos Funcionais - Classificação
	movimentoPistao : empurrarCaixa;

	// Blocos Funcionais - Usinagem

	// Blocos Funcionais - Empacotamento
	empCNC : FB_MoveTo;
	posicionarEstPlas : posicionarEsteiraPlastico;
 	posicionarEstMetal : posicionarEsteiraMetal;
 	movPlas : moverPlastico;
 	movMetal : moverMetal;

END_VAR

//--------------------------------------------------------------------------------------------
//-------------------------------TRATAMENTO DE VARIÁVEIS--------------------------------------
//----------------------------------------INÍCIO----------------------------------------------

// Variáveis de lógica inversa
EMER := NOT(FIO.i_Emergencia);
STOP := NOT(FIO.i_Stop);
OP2 := NOT(FIO.i_RS1);
OP3 := NOT(FIO.i_RS2);

// Led dos botões
FIO.o_LedSPMais := FIO.i_SPMais;
FIO.o_LedSPMenos := FIO.i_SPMenos;
FIO.o_LedStart := FIO.i_Start;
FIO.o_LedStop := NOT(FIO.i_Stop);

//------------------------------------------FINAL---------------------------------------------
//-------------------------------TRATAMENTO DE VARIÁVEIS--------------------------------------
//--------------------------------------------------------------------------------------------

//--------------------------------------------------------------------------------------------
//----------------------------------LÓGICA DOS SENSORES---------------------------------------
//----------------------------------------INÍCIO----------------------------------------------

IF Maquina1 AND NOT Emergencia1 AND NOT esperaCla THEN // Se a máquina 1 estiver operando
	Timer_sc(IN:=NOT FIO.i_SC); // A entrada dos timers será o inverso dos sensores
	Timer_op1(IN:=NOT FIO.i_DS2); // Logo quando os sensores detectarem algo, os timers reiniciam
ELSE // Caso contrário, os timers permanecem inativos
	Timer_sc(IN:=FALSE);
	Timer_op1(IN:=FALSE);
END_IF;

IF Maquina2 AND NOT Emergencia2 THEN // Se a máquina 2 estiver operando
<<<<<<< HEAD:PLC_PRG (PRG).st
<<<<<<< HEAD:PLC_PRG (PRG).st
	Timer_op2(IN:=NOT OP2); // A entrada dos timers será o inverso dos sensores
	Timer_usi(IN:=NOT FIO.i_MachiningCenterIsBusy); // Logo quando os sensores detectarem algo, os timers reiniciam
ELSE // Caso contrário, os timers permanecem inativos
=======
	Timer_op2(IN:=NOT OP2);
	Timer_usi(IN:=NOT FIO.i_MachiningCenterIsBusy);
ELSE
>>>>>>> origin/main:PLC_PRG.st
=======
	Timer_op2(IN:=NOT OP2);
	Timer_usi(IN:=NOT FIO.i_MachiningCenterIsBusy);
ELSE
>>>>>>> 670f2d2 (Código funcionando 100% e com 100% de eficiência):PLC_PRG.st
	Timer_op2(IN:=FALSE);
	Timer_usi(IN:=FALSE);
END_IF;

IF Maquina3 AND NOT Emergencia3 THEN // Se a máquina 3 estiver operando
	Timer_op3(IN:=NOT OP3); // A entrada do timer será o inverso do sensor
ELSE // Caso contrário, os timers permanecem inativos
	Timer_op3(IN:=FALSE);
END_IF;

//------------------------------------------FINAL---------------------------------------------
//----------------------------------LÓGICA DOS SENSORES---------------------------------------
//--------------------------------------------------------------------------------------------

//--------------------------------------------------------------------------------------------
//----------------------------------MÁQUINAS DE ESTADO----------------------------------------
//----------------------------------------INÍCIO----------------------------------------------

//----------------------------------MÁQUINA CLASSIFICADORA------------------------------------
//----------------------------------------INÍCIO----------------------------------------------

CASE E_Cla OF
	0: // Estado ocioso
	// Ação oneshot
	IF NOT os_cla[E_Cla] THEN
		os_cla := os_reset;

		delayEstabilizarBalanca(IN := FALSE); // Reinicia o timer de delay da balança
		global.Fila_cla(clear := TRUE); // Limpa fila de dados
		global.Fila_cla(clear := FALSE);

		os_cla[E_Cla] := TRUE;
	END_IF

    // Ações
	FIO.o_E1          := FALSE; // Esteira 1 parada
	FIO.o_E_SP        := FALSE; // Esteira 2 parada
	FIO.o_C1          := FALSE; // Pistão retraído
	FIO.o_NumCaixas := 0;

	// Transições de estado
  	IF Maquina1 THEN // Se receber o sinal Maquina1, a máquina classificadora sai do ócio
		E_Cla := 1;
	END_IF;

	1: // Liga Esteira
	// Ação oneshot
	IF NOT os_cla[E_Cla] THEN
		os_cla := os_reset;

		os_cla[E_Cla] := TRUE;
	END_IF

	// Ações
	FIO.o_E1    := TRUE; // Deixa a esteira 1 ligada
	FIO.o_E_SP  := TRUE; // Deixa a esteira 2 ligada

	// Transições de estado
    IF FIO.i_DS2 THEN // Se o sensor óptico 1 detectar algo
		IF esperaCla THEN // A máquina espera caso a usinagem tenha pedido
			E_Cla := 7;
		ELSE // Senão vai para o estado de estabilizar o peso
			E_Cla := 2;
		END_IF;
	END_IF;

	2: // Espera estabilizar peso
	// Ação oneshot
	IF NOT os_cla[E_Cla] THEN
		os_cla := os_reset;

		os_cla[E_Cla] := TRUE;
	END_IF

  	// Ações
	delayEstabilizarBalanca(IN := TRUE); // Delay para estabilizar a balança
	FIO.o_E1         := FALSE; // Para a esteira 1
	FIO.o_E_SP       := FALSE; // Para a esteira 2

	// Transições de estado
    IF delayEstabilizarBalanca.Q THEN // Se o timer da balança der sinal
		IF esperaCla THEN // Ele espera caso a usinagem peça
			E_Cla := 7;
		ELSE // Senão segue pra classificação de caixa ou não caixa
			E_Cla := 3;
		END_IF;
		delayEstabilizarBalanca(IN := FALSE);
	END_IF;

	3: // Classificação Caixa ou não caixa
	// Ação oneshot
	IF NOT os_cla[E_Cla] THEN
		os_cla := os_reset;

		caixa := (FIO.i_SP < 300); // Com a ação oneshot, determina se é uma caixa ou não pelo peso

		os_cla[E_Cla] := TRUE;
	END_IF

  	// Ações
	FIO.o_E1 := TRUE; // Esteira 1 ligada
	FIO.o_E_SP := FALSE; // Esteira da balança desligada

	// Transições de estado
    IF caixa THEN // Se for uma caixa passa para o estado de caixa detectada
		E_Cla := 4;
	ELSE // Se não for, passa para o estado de caixa não detectada
		E_Cla := 5;
	END_IF;

	4: // Caixa detectada
	// Ação oneshot
	IF NOT os_cla[E_Cla] THEN
		os_cla := os_reset;

		global.Fila_cla(pop := TRUE); // Na ação oneshot dá um pop na fila de classificação
		global.Fila_cla(pop := FALSE);

		os_cla[E_Cla] := TRUE;
	END_IF

  	// Ações
	FIO.o_E1 := TRUE; // Esteira 1 ligada
	FIO.o_E_SP := FALSE; // Esteira da balança desligada
	movimentoPistao(start:=TRUE); // Inicia o movimento do pistão

	// Transições de estado
<<<<<<< HEAD:PLC_PRG (PRG).st
    IF movimentoPistao.done THEN // Quando o movimento do pistão é concluído
		FIO.o_NumCaixas := FIO.o_NumCaixas + 1; // Aumenta a quantidade de caixas processadas
		IF esperaCla THEN // E espera caso a usinagem peça
=======
    IF movimentoPistao.done THEN
		FIO.o_NumCaixas := FIO.o_NumCaixas + 1;
		IF esperaCla THEN
>>>>>>> origin/main:PLC_PRG.st
			E_Cla := 7;
		ELSE // Caso não peça volta pro primeiro estado
			E_Cla := 1;
		END_IF;
		movimentoPistao(start:=FALSE);
	END_IF;

	5: // Caixa não detectada
	// Ação oneshot
	IF NOT os_cla[E_Cla] THEN
		os_cla := os_reset;

		pushFilaUsi(); // Na ação oneshot, usa a função pushFilaUsi, que tira o item da fila de
					   // classificação e manda para a fila de usinagem
		contador_classificacao := contador_classificacao + 1; // Aumenta a contagem dos itens que passaram
															  // na classificação

		os_cla[E_Cla] := TRUE;
	END_IF

  	// Ações
	FIO.o_E1 := TRUE; // Liga a esteira 1
	FIO.o_E_SP := TRUE; // Liga a esteira da balança

	// Transições de estado
    IF NOT FIO.i_DS2 THEN // Se não detectar mais com o sensor óptico
		IF esperaCla THEN // Espera caso a usinagem peça para esperar
			E_Cla := 7;
		ELSE // Caso contrário volta ao primeiro estado
			E_Cla := 1;
		END_IF;
	END_IF;

  	6: // Estado Emergência
	// Ação oneshot
	IF NOT os_cla[E_Cla] THEN
		os_cla := os_reset;

		global.Fila_cla(clear := TRUE); // Limpa a fila com uma ação oneshot
		global.Fila_cla(clear := FALSE);

		os_cla[E_Cla] := TRUE;
	END_IF

  	// Ações
<<<<<<< HEAD:PLC_PRG (PRG).st
	FIO.o_E1          	:= FALSE; // Desliga a esteira 1
	FIO.o_E_SP          := FALSE; // Desliga a esteira da balança
	FIO.o_C1           	:= FALSE; // Desliga o pistão
	FIO.o_NumCaixas 	:= 0; // Reseta o número de caixas processadas
	delayEstabilizarBalanca(IN := FALSE); // Reseta o timer de delay da balança
=======
	FIO.o_E1          := FALSE;
	FIO.o_E_SP          := FALSE;
	FIO.o_C1           := FALSE;
	FIO.o_NumCaixas := 0;
	delayEstabilizarBalanca(IN := FALSE);
>>>>>>> origin/main:PLC_PRG.st

	// Transições de estado

	7: // Espera
	// Ação oneshot
	IF NOT os_cla[E_Cla] THEN
		os_cla := os_reset;

		os_cla[E_Cla] := TRUE;
	END_IF

  	// Ações
	FIO.o_E1          := FALSE; // Desliga a esteira 1
	FIO.o_E_SP        := FALSE; // Desliga a esteira da balança
	delayEstabilizarBalanca(IN := FALSE); // Reseta o timer de delay da balança

	// Transições de estado
	IF NOT esperaCla THEN // Caso a usinagem não peça mais pra esperar a máquina volta ao estado anterior
		E_Cla := E_Cla_anterior;
	END_IF;

	ELSE // Caso a máquina não esteja em nenhum estado válido, ela retorna ao estado ocioso
		E_Cla := 0;

END_CASE;

// Transições de estado universais
IF Emergencia1 THEN
	E_Cla := 6;

ELSIF NOT(Maquina1) THEN
	E_Cla := 0;

END_IF;

// Ações Stateless

// Se der um rising no sensor capacitivo, ele registra o item na fila de classificação
trigSC(CLK := FIO.i_SC);
IF trigSC.Q THEN
	registrarItem();
END_IF;

//------------------------------------------FINAL---------------------------------------------
//----------------------------------MÁQUINA CLASSIFICADORA------------------------------------

//-----------------------------------MÁQUINA USINAGEM-----------------------------------------
//----------------------------------------INÍCIO----------------------------------------------

CASE E_Usi OF
	0: // Estado ocioso
	// Ação oneshot
	IF NOT os_usi[E_Usi] THEN
		os_usi := os_reset;

		global.Fila_usi(clear := TRUE); // Limpa fila
		global.Fila_usi(clear := FALSE);

		os_usi[E_Usi] := TRUE;
	END_IF

  	// Ações
	FIO.o_E2     := FALSE; // Esteira 2 desligada
	FIO.o_MachiningCenterProduceLids := FALSE; // Seta a máquina para não produzir tampas
	FIO.o_RB1_Reset := TRUE; // Reseta o robô
	FIO.o_RB1_Stop := FALSE; // Impede o robô travado
	FIO.o_RB1_Start := FALSE; // Impede o robô iniciar o movimento

	// Transições de estado
    IF Maquina2 THEN // Se a máquina supervisora mandar o sinal de ligar, a máquina de usinagem sai do ócio
		E_Usi := 1;
	END_IF;

	1: // Liga Esteira
	// Ação oneshot
	IF NOT os_usi[E_Usi] THEN
		os_usi := os_reset;

		os_usi[E_Usi] := TRUE;
	END_IF

  	// Ações
	FIO.o_E2 := TRUE; // Liga a esteira
	FIO.o_RB1_Reset := FALSE; // Impede o robô de resetar
	FIO.o_RB1_Stop := TRUE; // Deixa o robô travado
	FIO.o_RB1_Start := FALSE; // Impede o robô iniciar o movimento

	// Transições de estado
    IF OP2 THEN // Se o sensor optíco 2 detectar a peça, passa para o próximo estado
		E_Usi := 2;
	END_IF;

	2: // Usinagem
	// Ação oneshot
	IF NOT os_usi[E_Usi] THEN
		os_usi := os_reset;

		os_usi[E_Usi] := TRUE;
	END_IF

  	// Ações
	FIO.o_E2 := TRUE; // Liga a esteira
	// Se o item for metal, ele recebe o design fundo, se for plástico recebe o design de tampa
	FIO.o_MachiningCenterProduceLids := NOT(global.Fila_usi.itemOut.metal);
	FIO.o_RB1_Reset := FALSE; // Impede o robô de resetar
	FIO.o_RB1_Stop := FALSE; // Impede o robô travado
	FIO.o_RB1_Start := TRUE; // Inicia o movimento do robô

	// Transições de estado
	trigUsiConcluida(CLK:=FIO.i_MachiningCenterIsBusy);
  	IF trigUsiConcluida.Q THEN // Se a usinagem for concluída, passa pro próximo estado
		E_Usi := 3; // Volta pro estado 1
		contador_usinagem := contador_usinagem + 1; // Aumenta em um o números de coisas usinadas
		trigUsiConcluida(CLK:=FIO.i_MachiningCenterIsBusy);
	END_IF;

	3: // Passar item para a próxima fila
	// Ação oneshot
	IF NOT os_usi[E_Usi] THEN
		os_usi := os_reset;

		pushFilaEmp(); // Na ação oneshot, usa a função pushFilaEmp, que tira o item da fila de
					   // usinagem e manda para a fila de classificação

		os_usi[E_Usi] := TRUE;
	END_IF

  	// Ações
	FIO.o_E2 := FALSE; // Desliga a esteira
	FIO.o_RB1_Reset := FALSE; // Impede o robô de resetar
	FIO.o_RB1_Stop := FALSE; // Impede o robô travado
	FIO.o_RB1_Start := FALSE; // Impede o movimento do robô

	// Transições de estado
	E_Usi := 1; // Volta pro estado 1

  	4: // Estado Emergência
  	// Ação oneshot
	IF NOT os_usi[E_Usi] THEN
		os_usi := os_reset;

		global.Fila_usi(clear := TRUE); // Limpa a fila
		global.Fila_usi(clear := FALSE);

		os_usi[E_Usi] := TRUE;
	END_IF

  	// Ações
	FIO.o_E2     := FALSE; // Desliga a esteira
	FIO.o_RB1_Reset := FALSE; // Impede o robô de resetar
	FIO.o_RB1_Stop := TRUE; // Deixa o robô travado
	FIO.o_RB1_Start := FALSE; // Impede o robô iniciar o movimento

	ELSE // Caso a máquina não esteja em nenhum estado válido, ela retorna ao estado ocioso
		E_Usi := 0;

END_CASE;

// Transições de estado universais
IF Emergencia2 THEN
	E_Usi := 4;

ELSIF NOT(Maquina2) THEN
	E_Usi := 0;

END_IF;

// Ações Stateless

// Se a máquina de usinagem estiver ocupada e tiver item chegando ela faz as esteiras pararem
trigUsiOcupada(CLK:=FIO.i_MachiningCenterIsBusy AND OP2);
IF (FIO.i_MachiningCenterIsBusy AND OP2) THEN
	IF trigUsiOcupada.Q THEN // Se a máquina de usinagem acabou de ficar ocupada, ela salva o estado
							 // atual da máquina de classificação antes de pedir para esperar
		E_Cla_anterior := E_Cla;
	END_IF;
	trigUsiOcupada(CLK:=FIO.i_MachiningCenterIsBusy AND OP2);
	FIO.o_E2 := FALSE; // Desliga a esteira que leva até a usinagem
	esperaCla := TRUE; // Liga o sinal de espera da classificação, ou seja, pede para a classificação esperar
ELSE
	esperaCla := FALSE; // Caso a usinagem não esteja ocupada, não pede para a classificação parar
END_IF;

//------------------------------------------FINAL---------------------------------------------
//------------------------------------MÁQUINA USINAGEM----------------------------------------

//---------------------------------MÁQUINA EMPACOTAMENTO--------------------------------------
//----------------------------------------INÍCIO----------------------------------------------

CASE E_Emp OF
	0: // Estado ocioso
  	// Ação oneshot
	IF NOT os_emp[E_Emp] THEN
		os_emp := os_reset;

		global.Fila_emp(clear := TRUE); // Limpa a fila de empacotamento
		global.Fila_emp(clear := FALSE);

		os_emp[E_Emp] := TRUE;
	END_IF
  	// Ações
	// Seta o gantry para ficar na posição de ócio
	empCNC(targetX := constante.Xidle, targetY := constante.Yidle, targetZ := constante.Zidle, start := TRUE);
	FIO.o_E3          := FALSE; // Desliga a esteira que leva ao gantry
	FIO.o_EPLASTIC1 := FALSE; // Desliga as esteiras dos itens de plástico
	FIO.o_EPLASTIC2 := FALSE;
	FIO.o_EPLASTIC3 := FALSE;
	FIO.o_EMETAL1 := FALSE; // Desliga as esteiras dos itens de metal
	FIO.o_EMETAL2 := FALSE;
	FIO.o_EMETAL3 := FALSE;
	metal_counter := 0;
	plastico_counter := 0;
<<<<<<< HEAD:PLC_PRG (PRG).st
	FIO.o_NumPlastico := 0;
	FIO.o_NumMetal := 0;
=======
>>>>>>> edf0396 (Update PLC_PRG.st):PLC_PRG.st

	// Transições de estado
  	IF Maquina3 THEN // Se a máquina supervisora mandar o sinal de ligar, a máquina de empacotamento sai do ócio
		empCNC(start := FALSE);
		E_Emp := 1;
	END_IF;

	1: // Posicionar esteira de plástico
	// Ação oneshot
	IF NOT os_emp[E_Emp] THEN
		os_emp := os_reset;

		os_emp[E_Emp] := TRUE;
	END_IF

	// Ações
	FIO.o_E3 := FALSE; // Desliga a esteira que leva ao gantry
	posicionarEstPlas(start:=TRUE); // Inicia o FB que posiciona a caixa das esteiras de plástico

	// Transições de estado
	IF posicionarEstPlas.done THEN // Quando o posicionamento é concluído passa para o próximo estado
		posicionarEstPlas(start := FALSE);
		E_Emp := 2;
	END_IF;

	2: // Posicionar esteira de metal
	// Ação oneshot
	IF NOT os_emp[E_Emp] THEN
		os_emp := os_reset;

		os_emp[E_Emp] := TRUE;
	END_IF

  	// Ações
	FIO.o_E3 := FALSE; // Desliga a esteira que leva ao gantry
	posicionarEstMetal(start:=TRUE); // Inicia o FB que posiciona a caixa das esteiras de plástico

	// Transições de estado
	IF posicionarEstMetal.done THEN // Quando o posicionamento é concluído passa para o próximo estado
		posicionarEstMetal(start := FALSE);
		E_Emp := 3;
	END_IF;

	3: // Ligar esteira
	// Ação oneshot
	IF NOT os_emp[E_Emp] THEN
		os_emp := os_reset;

		os_emp[E_Emp] := TRUE;
	END_IF

  	// Ações
	FIO.o_E3 := TRUE; // Liga a esteira que leva ao gantry
	FIO.o_EPLASTIC1 := FALSE; // Desliga as esteiras dos itens de plástico
	FIO.o_EPLASTIC2 := FALSE;
	FIO.o_EPLASTIC3 := FALSE;
	FIO.o_EMETAL1 := FALSE; // Desliga as esteiras dos itens de metal
	FIO.o_EMETAL2 := FALSE;
	FIO.o_EMETAL3 := FALSE;

	// Transições de estado
	IF OP3 THEN // Caso o sensor óptico da esteira do empacotamento detecte algo
		IF global.Fila_emp.itemOut.metal THEN // Vai para o estado 5 se o último item da fila for metal
			E_Emp := 5;

		ELSE // Caso contrário vai para o estado 4
			E_Emp := 4;
		END_IF;

	END_IF;

	4: // Mover plástico
	// Ação oneshot
	IF NOT os_emp[E_Emp] THEN
		os_emp := os_reset;

		os_emp[E_Emp] := TRUE;
	END_IF

  	// Ações
	movPlas(start:=TRUE); // Inicia o FB de empacotar o item de plástico
	FIO.o_EPLASTIC1 := FALSE; // Desliga as esteiras dos itens de plástico
	FIO.o_EPLASTIC2 := FALSE;
	FIO.o_EPLASTIC3 := FALSE;
	FIO.o_EMETAL1 := FALSE; // Desliga as esteiras dos itens de metal
	FIO.o_EMETAL2 := FALSE;
	FIO.o_EMETAL3 := FALSE;

	// Transições de estado
	IF movPlas.done THEN // Quando o empacotamento é concluído
		global.Fila_emp(pop := TRUE); // Dá um pop na fila de empacotamento
		global.Fila_emp(pop := FALSE);
		movPlas(start := FALSE);
<<<<<<< HEAD:PLC_PRG (PRG).st
		FIO.o_NumPlastico := FIO.o_NumPlastico + 1; // Aumenta o contador de itens totais de plástico em 1
		plastico_counter := plastico_counter + 1; // Aumenta o contador de itens da caixa atual de plástico em 1
   		IF plastico_counter < itemPorCaixa THEN // Caso o contador de itens de plástico da caixa atual for
												// menor que os itens por caixa, volta pro estado 3
=======
		FIO.o_NumPlastico := FIO.o_NumPlastico + 1;
		plastico_counter := plastico_counter + 1;
   		IF plastico_counter < itemPorCaixa THEN
>>>>>>> origin/main:PLC_PRG.st
    		E_Emp := 3;

   		ELSE // Caso contrário, vai para o estado 6
    		E_Emp := 6;
   		END_IF;
  	END_IF;

  	5: // Mover metal
	// Ação oneshot
	IF NOT os_emp[E_Emp] THEN
		os_emp := os_reset;

		os_emp[E_Emp] := TRUE;
	END_IF

	// Ações
	movMetal(start:=TRUE); // Inicia o FB de empacotar o item de metal
	FIO.o_EPLASTIC1 := FALSE; // Desliga as esteiras dos itens de plástico
	FIO.o_EPLASTIC2 := FALSE;
	FIO.o_EPLASTIC3 := FALSE;
	FIO.o_EMETAL1 := FALSE; // Desliga as esteiras dos itens de metal
	FIO.o_EMETAL2 := FALSE;
	FIO.o_EMETAL3 := FALSE;

	// Transições de estado
  	IF movMetal.done THEN // Quando o empacotamento é concluído
		global.Fila_emp(pop := TRUE); // Dá um pop na fila de empacotamento
		global.Fila_emp(pop := FALSE);
   		movMetal(start := FALSE);
<<<<<<< HEAD:PLC_PRG (PRG).st
		FIO.o_NumMetal := FIO.o_NumMetal + 1; // Aumenta o contador de itens totais de metal em 1
   		metal_counter := metal_counter + 1; // Aumenta o contador de itens da caixa atual de metal em 1
   		IF metal_counter < itemPorCaixa THEN // Caso o contador de itens de metal da caixa atual for
    		E_Emp := 3;						 // menor que os itens por caixa, volta pro estado 3
   		ELSE // Caso contrário, vai para o estado 7
=======
		FIO.o_NumMetal := FIO.o_NumMetal + 1;
   		metal_counter := metal_counter + 1;
   		IF metal_counter < itemPorCaixa THEN
    		E_Emp := 3;
   		ELSE
>>>>>>> origin/main:PLC_PRG.st
    		E_Emp := 7;
   		END_IF;
  	END_IF;

  	6: // Mover esteira plástico
	// Ação oneshot
	IF NOT os_emp[E_Emp] THEN
		os_emp := os_reset;

		os_emp[E_Emp] := TRUE;
	END_IF

  	// Ações
	posicionarEstPlas(start:=TRUE); // Reposiciona a esteira de plástico para que outra caixa vazia fica em posição

	// Transições de estado
	IF posicionarEstPlas.done THEN // Caso a reposição da caixa for concluída
		posicionarEstPlas(start := FALSE);
		plastico_counter := 0; // Reseta o contador de itens da caixa atual de plástico
		E_Emp := 3; // E volta para o estado 3
	END_IF;

  	7: // Mover esteira metal
	// Ação oneshot
	IF NOT os_emp[E_Emp] THEN
		os_emp := os_reset;

		os_emp[E_Emp] := TRUE;
	END_IF

  	// Ações
  	posicionarEstMetal(start:=TRUE); // Reposiciona a esteira de metal para que outra caixa vazia fica em posição

	// Transições de estado
	IF posicionarEstMetal.done THEN // Caso a reposição da caixa for concluída
		posicionarEstMetal(start := FALSE);
		metal_counter := 0; // Reseta o contador de itens da caixa atual de metal
		E_Emp := 3; // E volta para o estado 3
	END_IF;

  	8: // Estado Emergência
  	// Ação oneshot
	IF NOT os_emp[E_Emp] THEN
		os_emp := os_reset;

		global.Fila_emp(clear:=TRUE); // Limpa a fila de empacotamento
		global.Fila_emp(clear:=FALSE);

		os_emp[E_Emp] := TRUE;
	END_IF
  	// Ações
	FIO.o_E3          := FALSE; // Desliga a esteira que leva ao empacotamento
	FIO.o_EPLASTIC1 := FALSE; // Desliga as esteiras dos itens de plástico
	FIO.o_EPLASTIC2 := FALSE;
	FIO.o_EPLASTIC3 := FALSE;
	FIO.o_EMETAL1 := FALSE; // Desliga as esteiras dos itens de metal
	FIO.o_EMETAL2 := FALSE;
	FIO.o_EMETAL3 := FALSE;
	metal_counter := 0;
	plastico_counter := 0;
<<<<<<< HEAD:PLC_PRG (PRG).st
	FIO.o_NumPlastico := 0;
	FIO.o_NumMetal := 0;
=======

>>>>>>> edf0396 (Update PLC_PRG.st):PLC_PRG.st

	ELSE // Caso a máquina não esteja em nenhum estado válido, ela retorna ao estado ocioso
		E_Emp := 0;

END_CASE;

// Transições de estado universais
IF Emergencia3 THEN
	E_Emp := 8;

ELSIF NOT(Maquina3) THEN
	E_Emp := 0;

END_IF;

// Ações stateless
IF OP3 THEN
	FIO.o_E3 := FALSE; // Desliga a esteira caso algo item seja detectado
END_IF;

//------------------------------------------FINAL---------------------------------------------
//---------------------------------MÁQUINA EMPACOTAMENTO--------------------------------------

//----------------------------------MÁQUINA SUPERVISORA---------------------------------------
//----------------------------------------INÍCIO----------------------------------------------

CASE E_Sup OF
	0: // Estado ocioso
  	// Ações
	Maquina1    			:= FALSE; // Desliga a máquina 1
	Maquina2    			:= FALSE; // Desliga a máquina 2
	Maquina3    			:= FALSE; // Desliga a máquina 3
	Emergencia1 			:= FALSE; // Emergência da máquina 1 desligada
	Emergencia2 			:= FALSE; // Emergência da máquina 2 desligada
	Emergencia3 			:= FALSE; // Emergência da máquina 3 desligada
	FIO.o_LedR  			:= FALSE; // Desliga o led vermelho
	FIO.o_LedG  			:= FALSE; // Desliga o led verde
	FIO.o_LedY  			:= TRUE;  // Liga o led amarelo
	contador_classificacao 	:= 0;	  // Contador de itens processados pela máquina 1 resetado
	contador_usinagem 		:= 0;	  // Contador de itens processados pela máquina 2 resetado

	trigSPMais(CLK:=FIO.i_SPMais);
	IF trigSPMais.Q THEN // Caso o botão SP+ for clicado, a variável itemPorCaixa aumenta em 1
		itemPorCaixa := itemPorCaixa + 1;
		trigSPMais(CLK:=FIO.i_SPMais);
	END_IF;

	trigSPMenos(CLK:=FIO.i_SPMenos);
	IF trigSPMenos.Q THEN // Caso o botão SP- for clicado, a variável itemPorCaixa diminui em 1
		itemPorCaixa := itemPorCaixa - 1;
		trigSPMenos(CLK:=FIO.i_SPMenos);
	END_IF;

	// Transições de estado
  	IF FIO.i_Start THEN // Se o botão FIO.i_Start for pressionado, a máquina supervisora sai do ócio
		E_Sup := 1;
	END_IF;

	1: // Ligar máquina classificação
	// Ações
	Maquina1   	:= TRUE;  // Liga a máquina 1
	Maquina2   	:= FALSE; // Desliga a máquina 2
	Maquina3   	:= FALSE; // Desliga a máquina 3
	Emergencia1 := FALSE; // Emergência da máquina 1 desligada
	Emergencia2 := FALSE; // Emergência da máquina 2 desligada
	Emergencia3 := FALSE; // Emergência da máquina 3 desligada
	FIO.o_LedR 	:= FALSE; // Desliga o led vermelho
	FIO.o_LedG 	:= TRUE;  // Liga o led verde
	FIO.o_LedY 	:= FALSE; // Desliga o led amarelo

	// Transições de estado
  	IF (contador_classificacao > 0) THEN // Se o primeiro item passar por todas os estados da máquina classificadora, passa pro próximo estado
		E_Sup := 2;
	END_IF;

	2: // Ligar máquina usinagem
  	// Ações
<<<<<<< HEAD:PLC_PRG (PRG).st
	Maquina1   	:= TRUE;  // Liga a máquina 1
	Maquina2   	:= TRUE;  // Liga a máquina 2
	Maquina3   	:= FALSE; // Desliga a máquina 3
	Emergencia1 := FALSE; // Emergência da máquina 1 desligada
	Emergencia2 := FALSE; // Emergência da máquina 2 desligada
	Emergencia3 := FALSE; // Emergência da máquina 3 desligada
	FIO.o_LedR 	:= FALSE; // Desliga o led vermelho
	FIO.o_LedG 	:= TRUE;  // Liga o led verde
	FIO.o_LedY 	:= FALSE; // Desliga o led amarelo
=======
	Maquina1   := TRUE;
	Maquina2   := TRUE;
	Maquina3   := FALSE;
	Emergencia1 := FALSE;
	Emergencia2 := FALSE;
	Emergencia3 := FALSE;
	FIO.o_LedR := FALSE;
	FIO.o_LedG := TRUE;
	FIO.o_LedY := FALSE;
>>>>>>> origin/main:PLC_PRG.st

	// Transições de estado
  	IF (contador_usinagem > 0) THEN // Se o primeiro item passar por todas os estados da máquina usinadora, passa pro próximo estado
		E_Sup := 3;
	END_IF;

	3: // Ligar máquina empacotamento
  	// Ações
	Maquina1   	:= TRUE;  // Liga a máquina 1
	Maquina2   	:= TRUE;  // Liga a máquina 2
	Maquina3   	:= TRUE;  // Liga a máquina 3
	Emergencia1 := FALSE; // Emergência da máquina 1 desligada
	Emergencia2 := FALSE; // Emergência da máquina 2 desligada
	Emergencia3 := FALSE; // Emergência da máquina 3 desligada
	FIO.o_LedR 	:= FALSE; // Desliga o led vermelho
	FIO.o_LedG 	:= TRUE;  // Liga o led verde
	FIO.o_LedY 	:= FALSE; // Desliga o led amarelo

	// Transições de estado

  	4: // Estado Emergência
  	// Ações
	Maquina1   				:= FALSE; // Desliga a máquina 1
	Maquina2   				:= FALSE; // Desliga a máquina 2
	Maquina3   				:= FALSE; // Desliga a máquina 3
	Emergencia1 			:= TRUE;  // Emergência da máquina 1 ligada
	Emergencia2 			:= TRUE;  // Emergência da máquina 2 ligada
	Emergencia3 			:= TRUE;  // Emergência da máquina 3 ligada
	FIO.o_LedR 				:= TRUE;  // Liga o led vermelho
	FIO.o_LedG 				:= FALSE; // Desliga o led verde
	FIO.o_LedY 				:= FALSE; // Desliga o led amarelo
	contador_classificacao 	:= 0;     // Contador de itens processados pela máquina 1 resetado
	contador_usinagem 		:= 0;     // Contador de itens processados pela máquina 2 resetado

	// Transições de estado

	ELSE // Caso a máquina não esteja em nenhum estado válido, ela retorna ao estado ocioso
		E_Sup := 0;

END_CASE;

// Transições de estado universais
<<<<<<< HEAD:PLC_PRG (PRG).st
<<<<<<< HEAD:PLC_PRG (PRG).st
IF (EMER OR Timer_sc.Q OR Timer_op1.Q OR Timer_op2.Q OR Timer_usi.Q OR Timer_op3.Q) THEN // Caso algum timer
																					// de sensor dispare
	E_Sup := 4; // Entra em estado de emergência
=======
=======
>>>>>>> 670f2d2 (Código funcionando 100% e com 100% de eficiência):PLC_PRG.st
IF (EMER OR Timer_sc.Q OR Timer_op1.Q OR Timer_op2.Q OR Timer_usi.Q OR Timer_op3.Q) THEN
	E_Sup := 4;
>>>>>>> origin/main:PLC_PRG.st

ELSIF STOP THEN // Caso o botão de parada for ativado, vai para o estado ocioso
	E_Sup := 0;

END_IF;

//------------------------------------------FINAL---------------------------------------------
//----------------------------------MÁQUINA SUPERVISORA---------------------------------------

//------------------------------------------FINAL---------------------------------------------
//-----------------------------------MÁQUINAS DE ESTADOS--------------------------------------
//--------------------------------------------------------------------------------------------

(* ---- PLC_PRG.st ---- *)
PROGRAM PLC_PRG
VAR
    // Estados das máquinas
    E_Cla : INT := 0;      // Classificadora
    E_Usi : INT := 0;      // Usinagem
    E_Emp : INT := 0;      // Empacotamento
    E_Sup : INT := 0;      // Supervisora

    // Entradas gerais
    START : BOOL;
    STOP  : BOOL;
	EMER  : BOOL;

    // Sinais de emergência
    Emergencia1 : BOOL := FALSE;
    Emergencia2 : BOOL := FALSE;
    Emergencia3 : BOOL := FALSE;

    // Comandos da máquina supervisora
    Maquina1 : BOOL := FALSE;   // Liga classificadora
    Maquina2 : BOOL := FALSE;   // Liga usinagem
    Maquina3 : BOOL := FALSE;   // Liga empacotamento

    // Sensores
    SC  : BOOL := FALSE;    // Sensor capacitivo
	SI  : BOOL := FALSE;    // Sensor indutivo
    OP1 : BOOL := FALSE;    // Sensor óptico 1
    OP2 : BOOL := FALSE;    // Sensor óptico 2
    OP3 : BOOL := FALSE;    // Sensor óptico 3

    // Contadores
    contador_classificacao : INT := 0;
    contador_usinagem      : INT := 0;

    // Contadores da empacotadora
    plastico_counter : INT := 0;
    metal_counter    : INT := 0;
    itemPorCaixa     : INT := 3;   // EXEMPLO — ajuste conforme sua lógica

    // Variáveis lógicas da empacotadora
    metal    : BOOL;
	caixa    : BOOL;

    // Variáveis da usinagem
    Mov1_concluido     : BOOL := FALSE;   // Movimento 1 concluído
    Mov2_concluido     : BOOL := FALSE;   // Movimento 2 concluído
    Usinagem_concluido : BOOL := FALSE;

	// Atuadores
	Esteira1 	  : BOOL := FALSE;
	Esteira2 	  : BOOL := FALSE;
	Esteira3 	  : BOOL := FALSE;
	Esteira4      : BOOL := FALSE;
	Esteira_plas  : BOOL := FALSE;
	Esteira_metal : BOOL := FALSE;
	Pistao1  	  : BOOL := FALSE;

	// Timers
	Timer_sc  	  : TON := (PT := T#30S);
	Timer_op1 	  : TON := (PT := T#30S);
	Timer_op2     : TON := (PT := T#30S);
	Timer_op3     : TON := (PT := T#30S);
	Timer_balanca : TON := (PT := T#2S);
	Timer_esteira : TON := (PT := T#3S);

	// Filas de itens
	Fila_cla : FB_PRODUCT_QUEUE;
	Fila_usi : FB_PRODUCT_QUEUE;
	Fila_emp : FB_PRODUCT_QUEUE;

	// Buffer de produto
	produtoBuffer : ST_PRODUCT;

	// Blocos Funcionais
	empCNC : FB_MoveTo;

END_VAR

//--------------------------------------------------------------------------------------------
//----------------------------------MÁQUINAS DE ESTADO----------------------------------------
//----------------------------------------INÍCIO----------------------------------------------

//----------------------------------MÁQUINA CLASSIFICADORA------------------------------------
//----------------------------------------INÍCIO----------------------------------------------

CASE E_Cla OF
	0: // Estado ocioso
    // Ações
	Esteira1          := FALSE;
	Esteira2          := FALSE;
	Pistao1           := FALSE;
	Timer_sc     (IN := FALSE);
	Timer_op1    (IN := FALSE);
	Timer_balanca(IN := FALSE);
	Fila_cla.clear    :=  TRUE;

	// Transições de estado
  	IF Maquina1 THEN // Se receber o sinal Maquina1, a máquina classificadora sai do ócio
		E_Cla := 1;
		Fila_cla.clear := FALSE;
	END_IF;

	1: // Liga Esteira
	// Ações
	Esteira1    := TRUE;
	Timer_sc(IN := TRUE);

	// Transições de estado
    IF SC THEN // Se o sensor capacitivo detectar algo, muda para o estado de classificação de metal
		E_Cla := 2;
	END_IF;

	2: // Classificação Metal ou não Metal
  	// Ações
	Timer_sc(IN := FALSE);
	Timer_op1(IN := TRUE);
	produtoBuffer.processed := FALSE;
	produtoBuffer.metal := SI;
	Fila_cla.itemIn := produtoBuffer;
	Fila_cla.push   := TRUE;

	// Transições de estado
    IF (NOT(SC) AND OP1) THEN // Se tanto o sensor capacitivo não detectar nada, quanto o sensor optíco 1 detectar, passa pro próximo estado
		E_Cla := 3;
		Fila_cla.push := FALSE;
	END_IF;

	3: // Espera estabilizar peso
  	// Ações
	Timer_op1.IN     := FALSE;
	Esteira1         := FALSE;
	Esteira2         := FALSE;
	Timer_balanca(IN := TRUE);

	// Transições de estado
    IF Timer_balanca.Q THEN // Se o timer 1 der sinal, passa pro próximo estado
		E_Cla := 4;
		Timer_balanca(IN := FALSE);
	END_IF;

	4: // Classificação Caixa ou não caixa
  	// Ações
	caixa := medirPeso();
	IF caixa THEN
		Pistao1 := TRUE;
	ELSE
		Pistao1 := FALSE;
		contador_classificacao := contador_classificacao + 1;
		IF (Fila_cla.itemOut <> 0) THEN
			Fila_usi.itemIn := Fila_cla.itemOut^;
			Fila_usi.push := TRUE;
		END_IF
	END_IF
	Fila_cla.pop := TRUE;

	// Transições de estado
    IF (NOT(OP1)) THEN // Se o sensor optíco 1 não detectar nada, volta ao início da operação
		E_Cla := 1;
		Fila_usi.push := FALSE;
	END_IF;

  	5: // Estado Emergência
  	// Ações
	Esteira1          := FALSE;
	Esteira2          := FALSE;
	Pistao1           := FALSE;
	Timer_sc     (IN := FALSE);
	Timer_op1    (IN := FALSE);
	Timer_balanca(IN := FALSE);
	Fila_cla.clear    :=  TRUE;

	// Transições de estado

	ELSE // Caso a máquina não esteja em nenhum estado válido, ela retorna ao estado ocioso
		E_Cla := 0;

END_CASE;

// Transições de estado universais
IF Emergencia1 THEN
	E_Cla := 5;

ELSIF NOT(Maquina1) THEN
	E_Cla := 0;

END_IF;
//------------------------------------------FINAL---------------------------------------------
//----------------------------------MÁQUINA CLASSIFICADORA------------------------------------

//-----------------------------------MÁQUINA USINAGEM-----------------------------------------
//----------------------------------------INÍCIO----------------------------------------------

CASE E_Usi OF
	0: // Estado ocioso
  	// Ações
	Esteira3     := FALSE;
	Timer_op2(IN := FALSE);
	interromperBraco();
	interromperUsinagem();
	Fila_usi.clear := TRUE;

	// Transições de estado
    IF Maquina2 THEN // Se a máquina supervisora mandar o sinal de ligar, a máquina de usinagem sai do ócio
		E_Usi := 1;
		Fila_usi.clear := FALSE;
	END_IF;

	1: // Liga Esteira
	// Ações
	Esteira3     := TRUE;
	Timer_op2(IN := TRUE);

	// Transições de estado
	IF NOT(Maquina2) THEN // Se a máquina supervisora mandar o sinal de desligar, a máquina de usinagem volta pro ócio
		E_Usi := 0;
    ELSIF OP2 THEN // Se o sensor optíco 2 detectar a peça, passa para o próximo estado
		E_Usi := 2;
	END_IF;

	2: // Pôr peça na usinagem
  	// Ações
	Timer_op2(IN := FALSE);
	Mov1();

	// Transições de estado
  	IF (Mov1_concluido) THEN // Se o movimento 1 do braço robótico for concluído, passa pro próximo estado
		E_Usi := 3;
	END_IF;

	3: // Usinagem
  	// Ações
	IF (Fila_usi.itemOut <> 0) THEN
		metal := Fila_usi.itemOut^.metal;
		IF metal THEN
			usinarMetal();
			Fila_usi.itemOut^ := TRUE;
		ELSE
			usinarPlastico();
			Fila_usi.itemOut^ := TRUE;
		END_IF;
	END_IF;

	// Transições de estado
  	IF (Usinagem_concluido) THEN // Se a usinagem for concluída, passa pro próximo estado
		E_Usi := 4;
	END_IF;

	4: // Tira peça da usinagem
  	// Ações
	Mov2();
	contador_usinagem := contador_usinagem + 1;
	IF (Fila_usi.itemOut <> 0) THEN
		Fila_emp.itemIn := Fila_usi.itemOut^;
		Fila_usi.pop := TRUE;
	END_IF;

	// Transições de estado
  	IF (Mov2_concluido) THEN // Se o movimento 2 do braço robótico for concluído, passa pro próximo estado
		E_Usi := 1;
		Fila_usi.pop := FALSE;
	END_IF;

  	5: // Estado Emergência
  	// Ações
	Esteira3     := FALSE;
	Timer_op2(IN := FALSE);
	interromperBraco();
	interromperUsinagem();
	Fila_usi.clear := TRUE;

	// Transições de estado

	ELSE // Caso a máquina não esteja em nenhum estado válido, ela retorna ao estado ocioso
		E_Usi := 0;

END_CASE;

// Transições de estado universais
IF Emergencia2 THEN
	E_Usi := 5;

ELSIF NOT(Maquina2) THEN
	E_Usi := 0;

END_IF;

//------------------------------------------FINAL---------------------------------------------
//------------------------------------MÁQUINA USINAGEM----------------------------------------

//---------------------------------MÁQUINA EMPACOTAMENTO--------------------------------------
//----------------------------------------INÍCIO----------------------------------------------

CASE E_Emp OF
	0: // Estado ocioso
  	// Ações
	Esteira4          := FALSE;
	Esteira_plas      := FALSE;
	Esteira_metal     := FALSE;
	Timer_op3(IN     := FALSE);
	Timer_esteira(IN := FALSE);
	Fila_emp.clear     := TRUE;

	// Transições de estado
  	IF Maquina3 THEN // Se a máquina supervisora mandar o sinal de ligar, a máquina de empacotamento sai do ócio
		E_Emp := 1;
		Fila_emp.clear := FALSE;
	END_IF;

	1: // Liga Esteira
	// Ações
	Esteira4       := TRUE;
	Esteira_plas  := FALSE;
	Esteira_metal := FALSE;
	Timer_op3(IN := TRUE);
	// Posicionar na esteira de plástico
	empCNC(targetX := 0, targetY := 5, targetZ := 5, start := TRUE);

	// Transições de estado
	IF NOT(Maquina3) THEN // Se a máquina supervisora mandar o sinal de desligar, a máquina de empacotamento volta pro ócio
		E_Emp := 0;
  	ELSIF OP3 THEN // Se o sensor optíco 3 detectar a peça, passa para o próximo estado
		E_Emp := 2;
	END_IF;

	2: // Pegar item
  	// Ações
    Esteira4      := FALSE;
	Timer_op3(IN := FALSE);
	// Pegar peça
	empCNC(targetX := 0, targetY := 5, targetZ := 10, start := TRUE);

	// Transições de estado
	IF empCNC.done THEN
		Succao := TRUE;
		IF (Fila_emp.itemOut <> 0) THEN
  			IF Fila_emp.itemOut^.metal THEN // Se o item pego for metal, segue pro estado 3
				E_Emp := 3;
			ELSE // Se não for, segue pro estado 4
				E_Emp := 4;
			END_IF;
		END_IF;
	END_IF;

	3: // Mover plástico
  	// Ações
	// Posicionar na esteira de plástico
	empCNC(targetX := 3, targetY := 5, targetZ := 10, start := TRUE);
  	Fila_emp.pop := TRUE;

	// Transições de estado
	IF empCNC.done THEN
		Succao := FALSE;
  		IF (plastico_counter < itemPorCaixa) THEN // Se a máquina supervisora mandar o sinal de ligar, a máquina de empacotamento sai do ócio
			plastico_counter := plastico_counter + 1;
			E_Emp := 1;
			Fila_emp.pop := FALSE;
		ELSE
			E_Emp := 5;
			Fila_emp.pop := FALSE;
		END_IF;
	END_IF;

	4: // Mover metal
  	// Ações
	// Posicionar na esteira de metal
	empCNC(targetX := 7, targetY := 5, targetZ := 10, start := TRUE);
  	Fila_emp.pop := TRUE;

	// Transições de estado
	IF empCNC.done THEN
		Succao := FALSE;
  		IF (metal_counter < itemPorCaixa) THEN // Se a máquina supervisora mandar o sinal de ligar, a máquina de empacotamento sai do ócio
			metal_counter := metal_counter + 1;
			E_Emp := 1;
		ELSE
			E_Emp := 6;
		END_IF;
	END_IF;

  	5: // Mover esteira plástico
  	// Ações
	Esteira_plas := TRUE;
	Timer_esteira(IN := TRUE);

	// Transições de estado
	IF Timer_esteira.Q THEN
  		E_Emp := 1;
	END_IF;

  	6: // Mover esteira metal
  	// Ações
	Esteira_metal := TRUE;
	Timer_esteira(IN := TRUE);

	// Transições de estado
  	IF Timer_esteira.Q THEN
  		E_Emp := 1;
	END_IF;

  	7: // Estado Emergência
  	// Ações
	Esteira4          := FALSE;
	Esteira_plas      := FALSE;
	Esteira_metal     := FALSE;
	Timer_op3(IN     := FALSE);
	Timer_esteira(IN := FALSE);
	Fila_emp.clear     := TRUE;

	// Transições de estado

	ELSE // Caso a máquina não esteja em nenhum estado válido, ela retorna ao estado ocioso
		E_Emp := 0;

END_CASE;

// Transições de estado universais
IF Emergencia3 THEN
	E_Emp := 7;

ELSIF NOT(Maquina3) THEN
	E_Emp := 0;

END_IF;

//------------------------------------------FINAL---------------------------------------------
//---------------------------------MÁQUINA EMPACOTAMENTO--------------------------------------

//----------------------------------MÁQUINA SUPERVISORA---------------------------------------
//----------------------------------------INÍCIO----------------------------------------------

CASE E_Sup OF
	0: // Estado ocioso
  	// Ações
	Maquina1    := FALSE;
	Maquina2    := FALSE;
	Maquina3    := FALSE;
	Emergencia1 := FALSE;
	Emergencia2 := FALSE;
	Emergencia3 := FALSE;

	// Transições de estado
  	IF START THEN // Se o botão start for pressionado, a máquina supervisora sai do ócio
		E_Sup := 1;
	END_IF;

	1: // Ligar máquina classificação
	// Ações
	Maquina1 := TRUE;

	// Transições de estado
  	IF (contador_classificacao > 0) THEN // Se o primeiro item passar por todas os estados da máquina classificadora, passa pro próximo estado
		E_Sup := 2;
	END_IF;

	2: // Ligar máquina usinagem
  	// Ações
	Maquina2 := TRUE;

	// Transições de estado
  	IF (contador_usinagem > 0) THEN // Se o primeiro item passar por todas os estados da máquina usinadora, passa pro próximo estado
		E_Sup := 3;
	END_IF;

	3: // Ligar máquina empacotamento
  	// Ações
	Maquina3 := TRUE;

	// Transições de estado

  	4: // Estado Emergência
  	// Ações
	Maquina1   := FALSE;
	Maquina2   := FALSE;
	Maquina3   := FALSE;
	Emergencia1 := TRUE;
	Emergencia2 := TRUE;
	Emergencia3 := TRUE;

	// Transições de estado

	ELSE // Caso a máquina não esteja em nenhum estado válido, ela retorna ao estado ocioso
		E_Sup := 0;

END_CASE;

// Transições de estado universais
IF (EMER OR Timer_sc.Q OR Timer_op1.Q OR Timer_op2.Q OR Timer_op3.Q) THEN
	E_Sup := 4;

ELSIF STOP THEN
	E_Sup := 0;

END_IF;

//------------------------------------------FINAL---------------------------------------------
//----------------------------------MÁQUINA SUPERVISORA---------------------------------------

//------------------------------------------FINAL---------------------------------------------
//-----------------------------------MÁQUINAS DE ESTADOS--------------------------------------
//--------------------------------------------------------------------------------------------

(* ---- PLC_PRG_VAR.st ---- *)
PROGRAM PLC_PRG
VAR
    // Estados das máquinas
    E_Cla : INT := 0;      // Classificadora
    E_Usi : INT := 0;      // Usinagem
    E_Emp : INT := 0;      // Empacotamento
    E_Sup : INT := 0;      // Supervisora

    // Entradas gerais
    START : BOOL;
    STOP  : BOOL;
	EMER  : BOOL;

    // Sinais de emergência
    Emergencia1 : BOOL := FALSE;
    Emergencia2 : BOOL := FALSE;
    Emergencia3 : BOOL := FALSE;

    // Comandos da máquina supervisora
    Maquina1 : BOOL := FALSE;   // Liga classificadora
    Maquina2 : BOOL := FALSE;   // Liga usinagem
    Maquina3 : BOOL := FALSE;   // Liga empacotamento

    // Sensores
    SC  : BOOL := FALSE;    // Sensor capacitivo
    OP1 : BOOL := FALSE;    // Sensor óptico 1
    OP2 : BOOL := FALSE;    // Sensor óptico 2
    OP3 : BOOL := FALSE;    // Sensor óptico 3

    // Temporizadores
    KT1 : BOOL := FALSE;    // Timer 1 pronto

    // Contadores
    contador_classificacao : INT := 0;
    contador_usinagem      : INT := 0;

    // Contadores da empacotadora
    plastico_counter : INT := 0;
    metal_counter    : INT := 0;
    itemPorCaixa     : INT := 3;   // EXEMPLO — ajuste conforme sua lógica

    // Variáveis lógicas da empacotadora
    metal    : BOOL;

    // Variáveis da usinagem
    Mov1_concluido     : BOOL := FALSE;   // Movimento 1 concluído
    Mov2_concluido     : BOOL := FALSE;   // Movimento 2 concluído
    Usinagem_concluido : BOOL := FALSE;

    // Contadores de erro
    Contador_sc  : BOOL := FALSE;
    Contador_op1 : BOOL := FALSE;
    Contador_op2 : BOOL := FALSE;
    Contador_op3 : BOOL := FALSE;
END_VAR
